KUKA KRL program: f1_Kuka_APT214T02S14.SRC

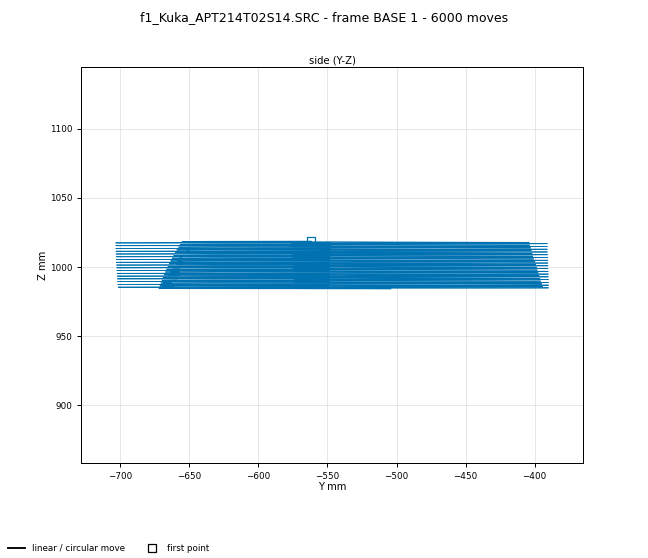
[picture p0: tool path of f1_Kuka_APT214T02S14.SRC in frame BASE 1, 6000 of 6001 moves have a stored position in this frame; points joined in program order, loops and branches not executed]
&ACCESS RVP
&REL 2
&PARAM TEMPLATE = C:\KRC\Roboter\Template\vorgabe
&PARAM EDITMASK = *
DEF f1_Kuka_APT214T02S14()


;FOLD INI;%{PE}%V3.2.0,%MKUKATPBASIS,%CINIT,%VCOMMON,%P
  ;FOLD BAS INI;%{E}%V3.2.0,%MKUKATPBASIS,%CINIT,%VINIT,%P
    GLOBAL INTERRUPT DECL 3 WHEN $STOPMESS==TRUE DO IR_STOPM ( )
    INTERRUPT ON 3
    BAS (#INITMOV,0 )
  ;ENDFOLD (BAS INI)
  ;FOLD USER INI;%{E}%V3.2.0,%MKUKATPUSER,%CINIT,%VINIT,%P
    ;Make your modifications here
  ;ENDFOLD (USER INI)
;ENDFOLD (INI)


;*** Make Null PTP Move
  PTP $pos_act

;*** Auto Load The Correct TOOL Data
  $tool=tool_data[2]

;*** Auto Load The Correct BASE Data
  $base=base_data[1]

  $ADVANCE = 5

;*** Restate Last Velocity
MMPM(30000.0)
SetRPM(8000)
LIN {X -0.057,Y -561.643,Z 1018.748,A 0.000,B 0.000,C 90.000,E1 350.679} C_DIS
LIN {X 0.006,Y -566.271,Z 1018.744,A 0.000,B 0.000,C 90.000,E1 349.982} C_DIS
LIN {X -0.209,Y -569.658,Z 1018.741,A 0.000,B 0.000,C 90.000,E1 349.454} C_DIS
LIN {X 0.145,Y -575.133,Z 1018.736,A 0.000,B 0.000,C 90.000,E1 348.465} C_DIS
LIN {X 0.098,Y -580.048,Z 1018.731,A 0.000,B 0.000,C 90.000,E1 347.521} C_DIS
LIN {X -0.016,Y -582.690,Z 1018.728,A 0.000,B 0.000,C 90.000,E1 346.992} C_DIS
LIN {X -0.106,Y -587.042,Z 1018.723,A 0.000,B 0.000,C 90.000,E1 346.061} C_DIS
LIN {X 0.162,Y -592.851,Z 1018.715,A 0.000,B 0.000,C 90.000,E1 344.700} C_DIS
LIN {X -0.022,Y -596.197,Z 1018.711,A 0.000,B 0.000,C 90.000,E1 343.921} C_DIS
LIN {X 0.114,Y -600.480,Z 1018.705,A 0.000,B 0.000,C 90.000,E1 342.851} C_DIS
LIN {X 0.194,Y -603.554,Z 1018.700,A 0.000,B 0.000,C 90.000,E1 342.054} C_DIS
LIN {X -0.152,Y -607.453,Z 1018.695,A 0.000,B 0.000,C 90.000,E1 341.040} C_DIS
LIN {X 0.011,Y -610.104,Z 1018.690,A 0.000,B 0.000,C 90.000,E1 340.242} C_DIS
LIN {X -0.056,Y -613.405,Z 1018.685,A 0.000,B 0.000,C 90.000,E1 339.209} C_DIS
LIN {X 0.142,Y -616.518,Z 1018.679,A 0.000,B 0.000,C 90.000,E1 338.156} C_DIS
LIN {X 0.387,Y -619.399,Z 1018.673,A 0.000,B 0.000,C 90.000,E1 337.102} C_DIS
LIN {X 0.107,Y -621.483,Z 1018.669,A 0.000,B 0.000,C 90.000,E1 336.357} C_DIS
LIN {X -0.153,Y -624.569,Z 1018.662,A 0.000,B 0.000,C 90.000,E1 335.101} C_DIS
LIN {X -0.110,Y -626.888,Z 1018.656,A 0.000,B 0.000,C 90.000,E1 334.076} C_DIS
LIN {X -0.009,Y -629.345,Z 1018.649,A 0.000,B 0.000,C 90.000,E1 332.794} C_DIS
LIN {X 0.070,Y -630.776,Z 1018.645,A 0.000,B 0.000,C 90.000,E1 332.025} C_DIS
LIN {X 0.010,Y -633.221,Z 1018.636,A 0.000,B 0.000,C 90.000,E1 330.511} C_DIS
LIN {X 0.149,Y -634.686,Z 1018.631,A 0.000,B 0.000,C 90.000,E1 329.488} C_DIS
LIN {X -0.103,Y -636.263,Z 1018.624,A 0.000,B 0.000,C 90.000,E1 328.250} C_DIS
LIN {X 0.259,Y -637.804,Z 1018.615,A 0.000,B 0.000,C 90.000,E1 326.707} C_DIS
LIN {X 0.039,Y -638.702,Z 1018.610,A 0.000,B 0.000,C 90.000,E1 325.722} C_DIS
LIN {X -0.035,Y -639.237,Z 1018.605,A 0.000,B 0.000,C 90.000,E1 324.975} C_DIS
LIN {X 0.163,Y -639.802,Z 1018.599,A 0.000,B 0.000,C 90.000,E1 323.703} C_DIS
LIN {X 0.259,Y -640.219,Z 1018.590,A 0.000,B 0.000,C 90.000,E1 322.190} C_DIS
LIN {X 0.161,Y -640.668,Z 1018.579,A 0.000,B 0.000,C 90.000,E1 320.194} C_DIS
LIN {X -0.417,Y -641.541,Z 1018.568,A 0.000,B 0.000,C 90.000,E1 318.243} C_DIS
LIN {X 0.035,Y -642.135,Z 1018.560,A 0.000,B 0.000,C 90.000,E1 316.701} C_DIS
LIN {X 0.325,Y -643.049,Z 1018.548,A 0.000,B 0.000,C 90.000,E1 314.676} C_DIS
LIN {X -0.126,Y -643.821,Z 1018.540,A 0.000,B 0.000,C 90.000,E1 313.218} C_DIS
LIN {X -0.031,Y -644.445,Z 1018.533,A 0.000,B 0.000,C 90.000,E1 311.962} C_DIS
LIN {X 0.052,Y -645.030,Z 1018.525,A 0.000,B 0.000,C 90.000,E1 310.458} C_DIS
LIN {X -0.187,Y -645.402,Z 1018.519,A 0.000,B 0.000,C 90.000,E1 309.483} C_DIS
LIN {X -0.007,Y -645.815,Z 1018.512,A 0.000,B 0.000,C 90.000,E1 308.222} C_DIS
LIN {X -0.130,Y -645.997,Z 1018.507,A 0.000,B 0.000,C 90.000,E1 307.237} C_DIS
LIN {X 0.087,Y -646.328,Z 1018.499,A 0.000,B 0.000,C 90.000,E1 305.724} C_DIS
LIN {X 0.403,Y -646.825,Z 1018.487,A 0.000,B 0.000,C 90.000,E1 303.706} C_DIS
LIN {X -0.135,Y -649.932,Z 1018.463,A 0.000,B 0.000,C 90.000,E1 299.283} C_DIS
LIN {X -0.198,Y -652.108,Z 1018.452,A 0.000,B 0.000,C 90.000,E1 297.308} C_DIS
LIN {X 0.032,Y -653.582,Z 1018.445,A 0.000,B 0.000,C 90.000,E1 296.052} C_DIS
LIN {X -0.122,Y -654.484,Z 1018.439,A 0.000,B 0.000,C 90.000,E1 295.079} C_DIS
LIN {X 0.046,Y -655.090,Z 1018.434,A 0.000,B 0.000,C 90.000,E1 294.079} C_DIS
LIN {X 0.223,Y -655.267,Z 1018.428,A 0.000,B 0.000,C 90.000,E1 293.078} C_DIS
LIN {X 0.259,Y -655.153,Z 1018.422,A 0.000,B 0.000,C 90.000,E1 291.844} C_DIS
LIN {X 0.363,Y -654.956,Z 1018.420,A 0.000,B 0.000,C 90.000,E1 291.589} C_DIS
LIN {X 0.327,Y -654.216,Z 1018.417,A 0.000,B 0.000,C 90.000,E1 291.099} C_DIS
LIN {X 0.287,Y -652.605,Z 1018.415,A 0.000,B 0.000,C 90.000,E1 290.610} C_DIS
LIN {X 0.150,Y -651.584,Z 1018.413,A 0.000,B 0.000,C 90.000,E1 290.375} C_DIS
LIN {X 0.238,Y -649.491,Z 1018.412,A 0.000,B 0.000,C 90.000,E1 290.120} C_DIS
LIN {X 0.095,Y -647.416,Z 1018.411,A 0.000,B 0.000,C 90.000,E1 289.885} C_DIS
LIN {X -0.373,Y -645.811,Z 1018.410,A 0.000,B 0.000,C 90.000,E1 289.758} C_DIS
LIN {X 0.299,Y -641.940,Z 1018.408,A 0.000,B 0.000,C 90.000,E1 289.450} C_DIS
LIN {X 0.228,Y -639.375,Z 1018.407,A 0.000,B 0.000,C 90.000,E1 289.268} C_DIS
LIN {X -0.172,Y -637.836,Z 1018.407,A 0.000,B 0.000,C 90.000,E1 289.214} C_DIS
LIN {X 0.150,Y -629.654,Z 1018.404,A 0.000,B 0.000,C 90.000,E1 288.779} C_DIS
LIN {X 0.077,Y -622.622,Z 1018.403,A 0.000,B 0.000,C 90.000,E1 288.489} C_DIS
LIN {X 0.244,Y -618.964,Z 1018.402,A 0.000,B 0.000,C 90.000,E1 288.308} C_DIS
LIN {X 0.190,Y -618.908,Z 1018.402,A 0.000,B 0.000,C 90.000,E1 288.308} C_DIS
LIN {X -0.227,Y -624.386,Z 1018.398,A 0.000,B 0.000,C 90.000,E1 287.583} C_DIS
LIN {X 0.131,Y -628.209,Z 1018.395,A 0.000,B 0.000,C 90.000,E1 287.040} C_DIS
LIN {X -0.090,Y -631.728,Z 1018.392,A 0.000,B 0.000,C 90.000,E1 286.551} C_DIS
LIN {X 0.134,Y -635.498,Z 1018.388,A 0.000,B 0.000,C 90.000,E1 285.898} C_DIS
LIN {X -0.045,Y -636.836,Z 1018.387,A 0.000,B 0.000,C 90.000,E1 285.662} C_DIS
LIN {X 0.224,Y -639.214,Z 1018.384,A 0.000,B 0.000,C 90.000,E1 285.134} C_DIS
LIN {X 0.059,Y -640.247,Z 1018.383,A 0.000,B 0.000,C 90.000,E1 284.898} C_DIS
LIN {X 0.359,Y -642.827,Z 1018.379,A 0.000,B 0.000,C 90.000,E1 284.120} C_DIS
LIN {X 0.204,Y -643.554,Z 1018.377,A 0.000,B 0.000,C 90.000,E1 283.883} C_DIS
LIN {X 0.050,Y -644.125,Z 1018.376,A 0.000,B 0.000,C 90.000,E1 283.647} C_DIS
LIN {X -0.251,Y -644.976,Z 1018.373,A 0.000,B 0.000,C 90.000,E1 283.175} C_DIS
LIN {X -0.065,Y -645.862,Z 1018.369,A 0.000,B 0.000,C 90.000,E1 282.411} C_DIS
LIN {X 0.140,Y -646.048,Z 1018.366,A 0.000,B 0.000,C 90.000,E1 281.895} C_DIS
LIN {X -0.148,Y -645.864,Z 1018.363,A 0.000,B 0.000,C 90.000,E1 281.422} C_DIS
LIN {X 0.044,Y -645.078,Z 1018.359,A 0.000,B 0.000,C 90.000,E1 280.658} C_DIS
LIN {X 0.261,Y -644.156,Z 1018.357,A 0.000,B 0.000,C 90.000,E1 280.141} C_DIS
LIN {X -0.048,Y -642.825,Z 1018.354,A 0.000,B 0.000,C 90.000,E1 279.670} C_DIS
LIN {X 0.161,Y -641.128,Z 1018.351,A 0.000,B 0.000,C 90.000,E1 279.151} C_DIS
LIN {X -0.004,Y -640.167,Z 1018.350,A 0.000,B 0.000,C 90.000,E1 278.916} C_DIS
LIN {X 0.191,Y -637.899,Z 1018.347,A 0.000,B 0.000,C 90.000,E1 278.398} C_DIS
LIN {X -0.258,Y -634.856,Z 1018.344,A 0.000,B 0.000,C 90.000,E1 277.936} C_DIS
LIN {X -0.158,Y -630.199,Z 1018.341,A 0.000,B 0.000,C 90.000,E1 277.296} C_DIS
LIN {X 0.115,Y -626.854,Z 1018.338,A 0.000,B 0.000,C 90.000,E1 276.891} C_DIS
LIN {X 0.180,Y -620.711,Z 1018.335,A 0.000,B 0.000,C 90.000,E1 276.258} C_DIS
LIN {X 0.086,Y -613.759,Z 1018.332,A 0.000,B 0.000,C 90.000,E1 275.682} C_DIS
LIN {X -0.147,Y -606.089,Z 1018.329,A 0.000,B 0.000,C 90.000,E1 275.163} C_DIS
LIN {X 0.078,Y -599.683,Z 1018.327,A 0.000,B 0.000,C 90.000,E1 274.759} C_DIS
LIN {X -0.286,Y -594.298,Z 1018.325,A 0.000,B 0.000,C 90.000,E1 274.531} C_DIS
LIN {X -0.227,Y -589.075,Z 1018.324,A 0.000,B 0.000,C 90.000,E1 274.302} C_DIS
LIN {X 0.101,Y -585.655,Z 1018.323,A 0.000,B 0.000,C 90.000,E1 274.131} C_DIS
LIN {X 0.250,Y -577.484,Z 1018.322,A 0.000,B 0.000,C 90.000,E1 273.898} C_DIS
LIN {X 0.081,Y -571.402,Z 1018.321,A 0.000,B 0.000,C 90.000,E1 273.784} C_DIS
LIN {X 0.255,Y -565.128,Z 1018.321,A 0.000,B 0.000,C 90.000,E1 273.669} C_DIS
LIN {X -0.046,Y -559.419,Z 1018.320,A 0.000,B 0.000,C 90.000,E1 273.669} C_DIS
LIN {X -0.087,Y -543.707,Z 1018.320,A 0.000,B 0.000,C 90.000,E1 273.669} C_DIS
LIN {X 0.158,Y -543.322,Z 1018.320,A 0.000,B 0.000,C 90.000,E1 273.555} C_DIS
LIN {X 0.168,Y -542.409,Z 1018.317,A 0.000,B 0.000,C 90.000,E1 273.037} C_DIS
LIN {X 0.219,Y -541.838,Z 1018.314,A 0.000,B 0.000,C 90.000,E1 272.465} C_DIS
LIN {X -0.138,Y -540.755,Z 1018.303,A 0.000,B 0.000,C 90.000,E1 270.516} C_DIS
LIN {X -0.051,Y -540.067,Z 1018.297,A 0.000,B 0.000,C 90.000,E1 269.370} C_DIS
LIN {X 0.022,Y -539.238,Z 1018.290,A 0.000,B 0.000,C 90.000,E1 268.224} C_DIS
LIN {X 0.136,Y -538.155,Z 1018.282,A 0.000,B 0.000,C 90.000,E1 266.788} C_DIS
LIN {X 0.202,Y -537.060,Z 1018.274,A 0.000,B 0.000,C 90.000,E1 265.355} C_DIS
LIN {X -0.198,Y -536.008,Z 1018.266,A 0.000,B 0.000,C 90.000,E1 263.970} C_DIS
LIN {X -0.075,Y -534.864,Z 1018.258,A 0.000,B 0.000,C 90.000,E1 262.527} C_DIS
LIN {X -0.027,Y -533.729,Z 1018.252,A 0.000,B 0.000,C 90.000,E1 261.376} C_DIS
LIN {X 0.162,Y -532.442,Z 1018.246,A 0.000,B 0.000,C 90.000,E1 260.208} C_DIS
LIN {X -0.122,Y -529.887,Z 1018.233,A 0.000,B 0.000,C 90.000,E1 257.937} C_DIS
LIN {X 0.163,Y -528.380,Z 1018.225,A 0.000,B 0.000,C 90.000,E1 256.464} C_DIS
LIN {X -0.113,Y -527.071,Z 1018.219,A 0.000,B 0.000,C 90.000,E1 255.338} C_DIS
LIN {X 0.112,Y -525.448,Z 1018.211,A 0.000,B 0.000,C 90.000,E1 253.866} C_DIS
LIN {X 0.089,Y -523.580,Z 1018.201,A 0.000,B 0.000,C 90.000,E1 252.127} C_DIS
LIN {X -0.103,Y -522.648,Z 1018.196,A 0.000,B 0.000,C 90.000,E1 251.275} C_DIS
LIN {X -0.173,Y -520.803,Z 1018.188,A 0.000,B 0.000,C 90.000,E1 249.826} C_DIS
LIN {X 0.037,Y -518.472,Z 1018.178,A 0.000,B 0.000,C 90.000,E1 248.050} C_DIS
LIN {X -0.090,Y -516.086,Z 1018.168,A 0.000,B 0.000,C 90.000,E1 246.305} C_DIS
LIN {X 0.166,Y -514.407,Z 1018.162,A 0.000,B 0.000,C 90.000,E1 245.101} C_DIS
LIN {X -0.062,Y -512.631,Z 1018.155,A 0.000,B 0.000,C 90.000,E1 243.948} C_DIS
LIN {X 0.143,Y -510.808,Z 1018.149,A 0.000,B 0.000,C 90.000,E1 242.743} C_DIS
LIN {X 0.149,Y -507.336,Z 1018.137,A 0.000,B 0.000,C 90.000,E1 240.667} C_DIS
LIN {X 0.050,Y -505.272,Z 1018.131,A 0.000,B 0.000,C 90.000,E1 239.488} C_DIS
LIN {X -0.134,Y -503.619,Z 1018.126,A 0.000,B 0.000,C 90.000,E1 238.614} C_DIS
LIN {X 0.136,Y -500.140,Z 1018.116,A 0.000,B 0.000,C 90.000,E1 236.786} C_DIS
LIN {X -0.092,Y -496.781,Z 1018.107,A 0.000,B 0.000,C 90.000,E1 235.308} C_DIS
LIN {X 0.047,Y -495.422,Z 1018.104,A 0.000,B 0.000,C 90.000,E1 234.689} C_DIS
LIN {X -0.260,Y -491.789,Z 1018.096,A 0.000,B 0.000,C 90.000,E1 233.210} C_DIS
LIN {X -0.041,Y -488.114,Z 1018.087,A 0.000,B 0.000,C 90.000,E1 231.662} C_DIS
LIN {X -0.062,Y -483.890,Z 1018.077,A 0.000,B 0.000,C 90.000,E1 229.828} C_DIS
LIN {X -0.319,Y -478.333,Z 1018.063,A 0.000,B 0.000,C 90.000,E1 227.391} C_DIS
LIN {X -0.011,Y -472.530,Z 1018.048,A 0.000,B 0.000,C 90.000,E1 224.555} C_DIS
LIN {X -0.056,Y -467.938,Z 1018.035,A 0.000,B 0.000,C 90.000,E1 222.366} C_DIS
LIN {X 0.069,Y -464.045,Z 1018.025,A 0.000,B 0.000,C 90.000,E1 220.458} C_DIS
LIN {X 0.019,Y -461.289,Z 1018.018,A 0.000,B 0.000,C 90.000,E1 219.197} C_DIS
LIN {X -0.075,Y -458.413,Z 1018.011,A 0.000,B 0.000,C 90.000,E1 217.935} C_DIS
LIN {X 0.041,Y -452.716,Z 1017.997,A 0.000,B 0.000,C 90.000,E1 215.358} C_DIS
LIN {X -0.070,Y -450.612,Z 1017.991,A 0.000,B 0.000,C 90.000,E1 214.405} C_DIS
LIN {X 0.126,Y -447.787,Z 1017.984,A 0.000,B 0.000,C 90.000,E1 213.086} C_DIS
LIN {X 0.095,Y -444.243,Z 1017.975,A 0.000,B 0.000,C 90.000,E1 211.465} C_DIS
LIN {X -0.058,Y -441.474,Z 1017.968,A 0.000,B 0.000,C 90.000,E1 210.178} C_DIS
LIN {X -0.062,Y -437.774,Z 1017.959,A 0.000,B 0.000,C 90.000,E1 208.537} C_DIS
LIN {X -0.126,Y -432.502,Z 1017.946,A 0.000,B 0.000,C 90.000,E1 206.232} C_DIS
LIN {X 0.073,Y -427.990,Z 1017.935,A 0.000,B 0.000,C 90.000,E1 204.207} C_DIS
LIN {X 0.168,Y -422.799,Z 1017.922,A 0.000,B 0.000,C 90.000,E1 201.844} C_DIS
LIN {X 0.122,Y -417.466,Z 1017.906,A 0.000,B 0.000,C 90.000,E1 199.141} C_DIS
LIN {X -0.105,Y -412.615,Z 1017.891,A 0.000,B 0.000,C 90.000,E1 196.441} C_DIS
LIN {X 0.195,Y -408.358,Z 1017.876,A 0.000,B 0.000,C 90.000,E1 193.647} C_DIS
LIN {X 0.070,Y -404.749,Z 1017.861,A 0.000,B 0.000,C 90.000,E1 190.894} C_DIS
LIN {X 0.084,Y -404.194,Z 1017.857,A 0.000,B 0.000,C 90.000,E1 190.197} C_DIS
LIN {X 0.093,Y -404.018,Z 1017.853,A 0.000,B 0.000,C 90.000,E1 189.500} C_DIS
LIN {X 0.097,Y -404.430,Z 1017.851,A 0.000,B 0.000,C 90.000,E1 189.151} C_DIS
LIN {X 0.192,Y -404.984,Z 1017.847,A 0.000,B 0.000,C 90.000,E1 188.454} C_DIS
LIN {X 0.198,Y -405.583,Z 1017.845,A 0.000,B 0.000,C 90.000,E1 188.106} C_DIS
LIN {X 0.121,Y -407.332,Z 1017.842,A 0.000,B 0.000,C 90.000,E1 187.530} C_DIS
LIN {X 0.118,Y -409.450,Z 1017.839,A 0.000,B 0.000,C 90.000,E1 187.011} C_DIS
LIN {X -0.044,Y -413.526,Z 1017.835,A 0.000,B 0.000,C 90.000,E1 186.258} C_DIS
LIN {X -0.010,Y -416.959,Z 1017.832,A 0.000,B 0.000,C 90.000,E1 185.739} C_DIS
LIN {X 0.062,Y -423.247,Z 1017.827,A 0.000,B 0.000,C 90.000,E1 184.878} C_DIS
LIN {X 0.138,Y -436.886,Z 1017.818,A 0.000,B 0.000,C 90.000,E1 183.212} C_DIS
LIN {X 0.195,Y -443.636,Z 1017.814,A 0.000,B 0.000,C 90.000,E1 182.407} C_DIS
LIN {X 0.161,Y -455.608,Z 1017.806,A 0.000,B 0.000,C 90.000,E1 180.974} C_DIS
LIN {X -0.192,Y -463.235,Z 1017.800,A 0.000,B 0.000,C 90.000,E1 180.057} C_DIS
LIN {X -0.229,Y -471.737,Z 1017.794,A 0.000,B 0.000,C 90.000,E1 178.969} C_DIS
LIN {X 0.081,Y -478.889,Z 1017.789,A 0.000,B 0.000,C 90.000,E1 177.993} C_DIS
LIN {X 0.129,Y -486.902,Z 1017.783,A 0.000,B 0.000,C 90.000,E1 176.906} C_DIS
LIN {X -0.153,Y -494.425,Z 1017.777,A 0.000,B 0.000,C 90.000,E1 175.869} C_DIS
LIN {X 0.120,Y -501.615,Z 1017.771,A 0.000,B 0.000,C 90.000,E1 174.780} C_DIS
LIN {X -0.177,Y -509.345,Z 1017.765,A 0.000,B 0.000,C 90.000,E1 173.628} C_DIS
LIN {X 0.106,Y -516.789,Z 1017.758,A 0.000,B 0.000,C 90.000,E1 172.413} C_DIS
LIN {X -0.007,Y -523.522,Z 1017.751,A 0.000,B 0.000,C 90.000,E1 171.254} C_DIS
LIN {X -0.241,Y -525.133,Z 1017.750,A 0.000,B 0.000,C 90.000,E1 171.027} C_DIS
LIN {X 0.004,Y -538.475,Z 1017.737,A 0.000,B 0.000,C 90.000,E1 168.701} C_DIS
LIN {X 0.212,Y -543.433,Z 1017.733,A 0.000,B 0.000,C 90.000,E1 167.825} C_DIS
LIN {X 0.271,Y -551.310,Z 1017.725,A 0.000,B 0.000,C 90.000,E1 166.408} C_DIS
LIN {X 0.072,Y -558.306,Z 1017.718,A 0.000,B 0.000,C 90.000,E1 165.172} C_DIS
LIN {X 0.123,Y -565.030,Z 1017.711,A 0.000,B 0.000,C 90.000,E1 163.921} C_DIS
LIN {X -0.219,Y -568.632,Z 1017.707,A 0.000,B 0.000,C 90.000,E1 163.268} C_DIS
LIN {X -0.290,Y -574.124,Z 1017.701,A 0.000,B 0.000,C 90.000,E1 162.181} C_DIS
LIN {X 0.079,Y -578.114,Z 1017.696,A 0.000,B 0.000,C 90.000,E1 161.329} C_DIS
LIN {X 0.075,Y -583.755,Z 1017.690,A 0.000,B 0.000,C 90.000,E1 160.115} C_DIS
LIN {X 0.212,Y -588.411,Z 1017.684,A 0.000,B 0.000,C 90.000,E1 159.028} C_DIS
LIN {X -0.040,Y -593.946,Z 1017.676,A 0.000,B 0.000,C 90.000,E1 157.720} C_DIS
LIN {X 0.080,Y -596.018,Z 1017.673,A 0.000,B 0.000,C 90.000,E1 157.177} C_DIS
LIN {X 0.276,Y -599.849,Z 1017.667,A 0.000,B 0.000,C 90.000,E1 156.102} C_DIS
LIN {X -0.198,Y -602.527,Z 1017.663,A 0.000,B 0.000,C 90.000,E1 155.357} C_DIS
LIN {X 0.037,Y -606.641,Z 1017.656,A 0.000,B 0.000,C 90.000,E1 154.024} C_DIS
LIN {X -0.204,Y -610.468,Z 1017.648,A 0.000,B 0.000,C 90.000,E1 152.743} C_DIS
LIN {X -0.066,Y -613.353,Z 1017.643,A 0.000,B 0.000,C 90.000,E1 151.691} C_DIS
LIN {X 0.097,Y -616.826,Z 1017.636,A 0.000,B 0.000,C 90.000,E1 150.383} C_DIS
LIN {X 0.072,Y -621.488,Z 1017.626,A 0.000,B 0.000,C 90.000,E1 148.584} C_DIS
LIN {X 0.150,Y -625.467,Z 1017.617,A 0.000,B 0.000,C 90.000,E1 147.041} C_DIS
LIN {X -0.231,Y -628.672,Z 1017.610,A 0.000,B 0.000,C 90.000,E1 145.801} C_DIS
LIN {X 0.165,Y -633.185,Z 1017.600,A 0.000,B 0.000,C 90.000,E1 143.989} C_DIS
LIN {X -0.240,Y -636.337,Z 1017.593,A 0.000,B 0.000,C 90.000,E1 142.763} C_DIS
LIN {X -0.088,Y -638.835,Z 1017.587,A 0.000,B 0.000,C 90.000,E1 141.743} C_DIS
LIN {X -0.007,Y -642.582,Z 1017.579,A 0.000,B 0.000,C 90.000,E1 140.231} C_DIS
LIN {X 0.054,Y -646.249,Z 1017.571,A 0.000,B 0.000,C 90.000,E1 138.728} C_DIS
LIN {X -0.024,Y -651.841,Z 1017.558,A 0.000,B 0.000,C 90.000,E1 136.500} C_DIS
LIN {X 0.151,Y -656.550,Z 1017.549,A 0.000,B 0.000,C 90.000,E1 134.757} C_DIS
LIN {X -0.043,Y -661.721,Z 1017.539,A 0.000,B 0.000,C 90.000,E1 133.056} C_DIS
LIN {X -0.081,Y -665.591,Z 1017.532,A 0.000,B 0.000,C 90.000,E1 131.838} C_DIS
LIN {X -0.047,Y -668.544,Z 1017.527,A 0.000,B 0.000,C 90.000,E1 130.862} C_DIS
LIN {X 0.030,Y -671.481,Z 1017.522,A 0.000,B 0.000,C 90.000,E1 129.886} C_DIS
LIN {X -0.262,Y -675.615,Z 1017.514,A 0.000,B 0.000,C 90.000,E1 128.463} C_DIS
LIN {X 0.028,Y -678.946,Z 1017.507,A 0.000,B 0.000,C 90.000,E1 127.237} C_DIS
LIN {X -0.014,Y -682.823,Z 1017.499,A 0.000,B 0.000,C 90.000,E1 125.804} C_DIS
LIN {X -0.010,Y -686.062,Z 1017.492,A 0.000,B 0.000,C 90.000,E1 124.612} C_DIS
LIN {X -0.176,Y -687.897,Z 1017.488,A 0.000,B 0.000,C 90.000,E1 123.913} C_DIS
LIN {X 0.113,Y -691.502,Z 1017.480,A 0.000,B 0.000,C 90.000,E1 122.467} C_DIS
LIN {X 0.090,Y -694.461,Z 1017.474,A 0.000,B 0.000,C 90.000,E1 121.288} C_DIS
LIN {X -0.117,Y -697.082,Z 1017.467,A 0.000,B 0.000,C 90.000,E1 120.129} C_DIS
LIN {X 0.046,Y -698.438,Z 1017.463,A 0.000,B 0.000,C 90.000,E1 119.411} C_DIS
LIN {X 0.147,Y -700.214,Z 1017.457,A 0.000,B 0.000,C 90.000,E1 118.231} C_DIS
LIN {X 0.342,Y -701.001,Z 1017.453,A 0.000,B 0.000,C 90.000,E1 117.513} C_DIS
LIN {X -0.307,Y -702.750,Z 1017.441,A 0.000,B 0.000,C 90.000,E1 115.463} C_DIS
LIN {X 0.237,Y -703.225,Z 1017.438,A 0.000,B 0.000,C 90.000,E1 114.719} C_DIS
LIN {X 0.158,Y -703.239,Z 1017.435,A 0.000,B 0.000,C 90.000,E1 114.259} C_DIS
LIN {X 0.150,Y -703.096,Z 1017.434,A 0.000,B 0.000,C 90.000,E1 114.027} C_DIS
LIN {X 0.065,Y -702.357,Z 1017.431,A 0.000,B 0.000,C 90.000,E1 113.567} C_DIS
LIN {X 0.061,Y -701.548,Z 1017.430,A 0.000,B 0.000,C 90.000,E1 113.334} C_DIS
LIN {X -0.315,Y -699.027,Z 1017.427,A 0.000,B 0.000,C 90.000,E1 112.898} C_DIS
LIN {X -0.183,Y -698.177,Z 1017.426,A 0.000,B 0.000,C 90.000,E1 112.770} C_DIS
LIN {X -0.051,Y -696.915,Z 1017.426,A 0.000,B 0.000,C 90.000,E1 112.642} C_DIS
LIN {X 0.256,Y -690.392,Z 1017.424,A 0.000,B 0.000,C 90.000,E1 112.206} C_DIS
LIN {X -0.206,Y -688.443,Z 1017.423,A 0.000,B 0.000,C 90.000,E1 112.153} C_DIS
LIN {X 0.230,Y -685.655,Z 1017.423,A 0.000,B 0.000,C 90.000,E1 112.025} C_DIS
LIN {X 0.192,Y -683.468,Z 1017.422,A 0.000,B 0.000,C 90.000,E1 111.972} C_DIS
LIN {X -0.229,Y -675.140,Z 1017.422,A 0.000,B 0.000,C 90.000,E1 111.897} C_DIS
LIN {X -0.243,Y -615.838,Z 1017.422,A 0.000,B 0.000,C 90.000,E1 111.897} C_DIS
LIN {X 0.286,Y -610.721,Z 1017.421,A 0.000,B 0.000,C 90.000,E1 111.716} C_DIS
LIN {X 0.239,Y -605.536,Z 1017.420,A 0.000,B 0.000,C 90.000,E1 111.535} C_DIS
LIN {X -0.193,Y -599.101,Z 1017.418,A 0.000,B 0.000,C 90.000,E1 111.280} C_DIS
LIN {X -0.045,Y -593.333,Z 1017.416,A 0.000,B 0.000,C 90.000,E1 110.918} C_DIS
LIN {X 0.263,Y -587.741,Z 1017.414,A 0.000,B 0.000,C 90.000,E1 110.482} C_DIS
LIN {X 0.180,Y -576.703,Z 1017.409,A 0.000,B 0.000,C 90.000,E1 109.577} C_DIS
LIN {X 0.101,Y -570.755,Z 1017.406,A 0.000,B 0.000,C 90.000,E1 109.141} C_DIS
LIN {X 0.059,Y -562.295,Z 1017.404,A 0.000,B 0.000,C 90.000,E1 108.671} C_DIS
LIN {X -0.267,Y -555.586,Z 1017.402,A 0.000,B 0.000,C 90.000,E1 108.362} C_DIS
LIN {X -0.040,Y -549.719,Z 1017.400,A 0.000,B 0.000,C 90.000,E1 108.000} C_DIS
LIN {X 0.141,Y -548.390,Z 1017.399,A 0.000,B 0.000,C 90.000,E1 107.819} C_DIS
LIN {X 0.099,Y -548.381,Z 1017.399,A 0.000,B 0.000,C 90.000,E1 107.819} C_DIS
LIN {X 0.096,Y -548.038,Z 1017.397,A 0.000,B 0.000,C 90.000,E1 107.402} C_DIS
LIN {X 0.126,Y -548.283,Z 1017.392,A 0.000,B 0.000,C 90.000,E1 106.567} C_DIS
LIN {X -0.047,Y -549.100,Z 1017.383,A 0.000,B 0.000,C 90.000,E1 104.898} C_DIS
LIN {X 0.021,Y -551.619,Z 1017.363,A 0.000,B 0.000,C 90.000,E1 101.243} C_DIS
LIN {X -0.218,Y -553.984,Z 1017.350,A 0.000,B 0.000,C 90.000,E1 99.029} C_DIS
LIN {X 0.065,Y -554.939,Z 1017.345,A 0.000,B 0.000,C 90.000,E1 98.163} C_DIS
LIN {X 0.113,Y -556.784,Z 1017.336,A 0.000,B 0.000,C 90.000,E1 96.486} C_DIS
LIN {X -0.063,Y -557.848,Z 1017.330,A 0.000,B 0.000,C 90.000,E1 95.391} C_DIS
LIN {X -0.271,Y -558.743,Z 1017.324,A 0.000,B 0.000,C 90.000,E1 94.302} C_DIS
LIN {X 0.217,Y -559.593,Z 1017.316,A 0.000,B 0.000,C 90.000,E1 92.865} C_DIS
LIN {X 0.217,Y -560.345,Z 1017.307,A 0.000,B 0.000,C 90.000,E1 91.203} C_DIS
LIN {X 0.225,Y -561.031,Z 1017.298,A 0.000,B 0.000,C 90.000,E1 89.542} C_DIS
LIN {X 0.163,Y -561.609,Z 1017.290,A 0.000,B 0.000,C 90.000,E1 88.165} C_DIS
LIN {X -0.009,Y -561.906,Z 1017.284,A 0.000,B 0.000,C 90.000,E1 87.078} C_DIS
LIN {X 0.065,Y -562.206,Z 1017.275,A 0.000,B 0.000,C 90.000,E1 85.412} C_DIS
LIN {X 0.199,Y -562.545,Z 1017.265,A 0.000,B 0.000,C 90.000,E1 83.742} C_DIS
LIN {X 0.104,Y -562.770,Z 1017.259,A 0.000,B 0.000,C 90.000,E1 82.648} C_DIS
LIN {X -0.085,Y -563.293,Z 1017.249,A 0.000,B 0.000,C 90.000,E1 80.735} C_DIS
LIN {X -0.002,Y -564.091,Z 1017.236,A 0.000,B 0.000,C 90.000,E1 78.522} C_DIS
LIN {X -0.118,Y -564.947,Z 1017.227,A 0.000,B 0.000,C 90.000,E1 76.881} C_DIS
LIN {X -0.157,Y -566.331,Z 1017.215,A 0.000,B 0.000,C 90.000,E1 74.685} C_DIS
LIN {X 0.060,Y -567.604,Z 1017.206,A 0.000,B 0.000,C 90.000,E1 73.015} C_DIS
LIN {X 0.129,Y -568.610,Z 1017.198,A 0.000,B 0.000,C 90.000,E1 71.638} C_DIS
LIN {X 0.010,Y -569.824,Z 1017.189,A 0.000,B 0.000,C 90.000,E1 70.007} C_DIS
LIN {X -0.079,Y -571.122,Z 1017.178,A 0.000,B 0.000,C 90.000,E1 68.103} C_DIS
LIN {X 0.076,Y -572.215,Z 1017.168,A 0.000,B 0.000,C 90.000,E1 66.177} C_DIS
LIN {X 0.129,Y -572.934,Z 1017.159,A 0.000,B 0.000,C 90.000,E1 64.537} C_DIS
LIN {X -0.064,Y -573.642,Z 1017.150,A 0.000,B 0.000,C 90.000,E1 62.922} C_DIS
LIN {X -0.237,Y -574.211,Z 1017.141,A 0.000,B 0.000,C 90.000,E1 61.307} C_DIS
LIN {X 0.032,Y -574.642,Z 1017.133,A 0.000,B 0.000,C 90.000,E1 59.921} C_DIS
LIN {X 0.306,Y -575.026,Z 1017.125,A 0.000,B 0.000,C 90.000,E1 58.535} C_DIS
LIN {X 0.369,Y -575.476,Z 1017.115,A 0.000,B 0.000,C 90.000,E1 56.628} C_DIS
LIN {X -0.161,Y -575.630,Z 1017.109,A 0.000,B 0.000,C 90.000,E1 55.595} C_DIS
LIN {X 0.262,Y -575.723,Z 1017.101,A 0.000,B 0.000,C 90.000,E1 54.196} C_DIS
LIN {X 0.215,Y -575.521,Z 1017.094,A 0.000,B 0.000,C 90.000,E1 52.844} C_DIS
LIN {X 0.007,Y -575.182,Z 1017.088,A 0.000,B 0.000,C 90.000,E1 51.778} C_DIS
LIN {X -0.299,Y -574.711,Z 1017.082,A 0.000,B 0.000,C 90.000,E1 50.723} C_DIS
LIN {X -0.026,Y -573.879,Z 1017.074,A 0.000,B 0.000,C 90.000,E1 49.337} C_DIS
LIN {X 0.030,Y -573.027,Z 1017.068,A 0.000,B 0.000,C 90.000,E1 48.243} C_DIS
LIN {X 0.379,Y -572.281,Z 1017.064,A 0.000,B 0.000,C 90.000,E1 47.391} C_DIS
LIN {X -0.092,Y -571.368,Z 1017.059,A 0.000,B 0.000,C 90.000,E1 46.620} C_DIS
LIN {X -0.177,Y -570.266,Z 1017.054,A 0.000,B 0.000,C 90.000,E1 45.810} C_DIS
LIN {X -0.272,Y -568.999,Z 1017.050,A 0.000,B 0.000,C 90.000,E1 45.000} C_DIS
LIN {X 0.017,Y -567.525,Z 1017.045,A 0.000,B 0.000,C 90.000,E1 44.150} C_DIS
LIN {X -0.017,Y -565.356,Z 1017.039,A 0.000,B 0.000,C 90.000,E1 43.056} C_DIS
LIN {X -0.136,Y -563.436,Z 1017.035,A 0.000,B 0.000,C 90.000,E1 42.243} C_DIS
LIN {X 0.108,Y -561.232,Z 1017.030,A 0.000,B 0.000,C 90.000,E1 41.391} C_DIS
LIN {X -0.131,Y -559.651,Z 1017.027,A 0.000,B 0.000,C 90.000,E1 40.862} C_DIS
LIN {X 0.066,Y -556.969,Z 1017.022,A 0.000,B 0.000,C 90.000,E1 40.011} C_DIS
LIN {X -0.054,Y -553.052,Z 1017.016,A 0.000,B 0.000,C 90.000,E1 38.910} C_DIS
LIN {X -0.286,Y -549.604,Z 1017.012,A 0.000,B 0.000,C 90.000,E1 38.096} C_DIS
LIN {X 0.065,Y -545.262,Z 1017.006,A 0.000,B 0.000,C 90.000,E1 37.076} C_DIS
LIN {X 0.170,Y -541.278,Z 1017.001,A 0.000,B 0.000,C 90.000,E1 36.217} C_DIS
LIN {X 0.068,Y -537.713,Z 1016.997,A 0.000,B 0.000,C 90.000,E1 35.518} C_DIS
LIN {X -0.068,Y -532.390,Z 1016.992,A 0.000,B 0.000,C 90.000,E1 34.532} C_DIS
LIN {X 0.166,Y -526.623,Z 1016.986,A 0.000,B 0.000,C 90.000,E1 33.499} C_DIS
LIN {X 0.205,Y -521.290,Z 1016.981,A 0.000,B 0.000,C 90.000,E1 32.625} C_DIS
LIN {X -0.080,Y -516.572,Z 1016.977,A 0.000,B 0.000,C 90.000,E1 31.926} C_DIS
LIN {X 0.029,Y -511.474,Z 1016.973,A 0.000,B 0.000,C 90.000,E1 31.180} C_DIS
LIN {X -0.174,Y -505.839,Z 1016.969,A 0.000,B 0.000,C 90.000,E1 30.463} C_DIS
LIN {X -0.040,Y -502.296,Z 1016.967,A 0.000,B 0.000,C 90.000,E1 30.001} C_DIS
LIN {X -0.243,Y -495.735,Z 1016.963,A 0.000,B 0.000,C 90.000,E1 29.283} C_DIS
LIN {X 0.300,Y -489.057,Z 1016.958,A 0.000,B 0.000,C 90.000,E1 28.487} C_DIS
LIN {X -0.303,Y -481.950,Z 1016.955,A 0.000,B 0.000,C 90.000,E1 27.847} C_DIS
LIN {X -0.114,Y -474.732,Z 1016.951,A 0.000,B 0.000,C 90.000,E1 27.129} C_DIS
LIN {X -0.065,Y -467.441,Z 1016.947,A 0.000,B 0.000,C 90.000,E1 26.437} C_DIS
LIN {X -0.132,Y -459.951,Z 1016.943,A 0.000,B 0.000,C 90.000,E1 25.771} C_DIS
LIN {X -0.031,Y -449.306,Z 1016.938,A 0.000,B 0.000,C 90.000,E1 24.847} C_DIS
LIN {X 0.109,Y -431.519,Z 1016.929,A 0.000,B 0.000,C 90.000,E1 23.281} C_DIS
LIN {X 0.162,Y -418.312,Z 1016.923,A 0.000,B 0.000,C 90.000,E1 22.025} C_DIS
LIN {X -0.032,Y -406.782,Z 1016.916,A 0.000,B 0.000,C 90.000,E1 20.844} C_DIS
LIN {X 0.060,Y -397.678,Z 1016.910,A 0.000,B 0.000,C 90.000,E1 19.758} C_DIS
LIN {X -0.150,Y -394.148,Z 1016.907,A 0.000,B 0.000,C 90.000,E1 19.268} C_DIS
LIN {X 0.112,Y -392.358,Z 1016.905,A 0.000,B 0.000,C 90.000,E1 18.852} C_DIS
LIN {X -0.179,Y -391.201,Z 1016.902,A 0.000,B 0.000,C 90.000,E1 18.362} C_DIS
LIN {X -0.084,Y -390.894,Z 1016.898,A 0.000,B 0.000,C 90.000,E1 17.638} C_DIS
LIN {X 0.064,Y -391.921,Z 1016.890,A 0.000,B 0.000,C 90.000,E1 16.205} C_DIS
LIN {X 0.145,Y -397.228,Z 1016.865,A 0.000,B 0.000,C 90.000,E1 11.591} C_DIS
LIN {X -0.034,Y -404.136,Z 1016.841,A 0.000,B 0.000,C 90.000,E1 7.409} C_DIS
LIN {X -0.135,Y -412.095,Z 1016.820,A 0.000,B 0.000,C 90.000,E1 3.612} C_DIS
LIN {X -0.119,Y -414.440,Z 1016.814,A 0.000,B 0.000,C 90.000,E1 2.579} C_DIS
LIN {X -0.113,Y -415.372,Z 1016.812,A 0.000,B 0.000,C 90.000,E1 2.236} C_DIS
LIN {X -0.083,Y -417.071,Z 1016.810,A 0.000,B 0.000,C 90.000,E1 1.718} C_DIS
LIN {X -0.096,Y -418.967,Z 1016.808,A 0.000,B 0.000,C 90.000,E1 1.375} C_DIS
LIN {X -0.140,Y -420.859,Z 1016.806,A 0.000,B 0.000,C 90.000,E1 1.088} C_DIS
LIN {X 0.203,Y -423.348,Z 1016.804,A 0.000,B 0.000,C 90.000,E1 0.745} C_DIS
LIN {X -0.201,Y -426.872,Z 1016.803,A 0.000,B 0.000,C 90.000,E1 0.516} C_DIS
LIN {X 0.135,Y -428.624,Z 1016.802,A 0.000,B 0.000,C 90.000,E1 0.344} C_DIS
LIN {X 0.166,Y -438.310,Z 1016.799,A 0.000,B 0.000,C 90.000,E1 359.771} C_DIS
LIN {X -0.002,Y -448.310,Z 1016.796,A 0.000,B 0.000,C 90.000,E1 359.198} C_DIS
LIN {X -0.135,Y -463.144,Z 1016.791,A 0.000,B 0.000,C 90.000,E1 358.339} C_DIS
LIN {X -0.158,Y -479.788,Z 1016.785,A 0.000,B 0.000,C 90.000,E1 357.364} C_DIS
LIN {X 0.124,Y -488.025,Z 1016.783,A 0.000,B 0.000,C 90.000,E1 356.849} C_DIS
LIN {X 0.064,Y -497.732,Z 1016.779,A 0.000,B 0.000,C 90.000,E1 356.274} C_DIS
LIN {X -0.069,Y -508.895,Z 1016.775,A 0.000,B 0.000,C 90.000,E1 355.584} C_DIS
LIN {X -0.205,Y -516.587,Z 1016.773,A 0.000,B 0.000,C 90.000,E1 355.065} C_DIS
LIN {X 0.108,Y -525.380,Z 1016.769,A 0.000,B 0.000,C 90.000,E1 354.375} C_DIS
LIN {X -0.073,Y -532.612,Z 1016.766,A 0.000,B 0.000,C 90.000,E1 353.799} C_DIS
LIN {X 0.028,Y -539.584,Z 1016.762,A 0.000,B 0.000,C 90.000,E1 353.166} C_DIS
LIN {X -0.072,Y -546.155,Z 1016.758,A 0.000,B 0.000,C 90.000,E1 352.527} C_DIS
LIN {X -0.030,Y -552.325,Z 1016.755,A 0.000,B 0.000,C 90.000,E1 351.837} C_DIS
LIN {X 0.205,Y -556.967,Z 1016.752,A 0.000,B 0.000,C 90.000,E1 351.254} C_DIS
LIN {X 0.141,Y -562.117,Z 1016.748,A 0.000,B 0.000,C 90.000,E1 350.566} C_DIS
LIN {X -0.104,Y -565.875,Z 1016.745,A 0.000,B 0.000,C 90.000,E1 350.038} C_DIS
LIN {X 0.238,Y -569.316,Z 1016.742,A 0.000,B 0.000,C 90.000,E1 349.454} C_DIS
LIN {X 0.009,Y -574.835,Z 1016.736,A 0.000,B 0.000,C 90.000,E1 348.522} C_DIS
LIN {X 0.186,Y -578.468,Z 1016.733,A 0.000,B 0.000,C 90.000,E1 347.825} C_DIS
LIN {X -0.155,Y -582.494,Z 1016.728,A 0.000,B 0.000,C 90.000,E1 347.048} C_DIS
LIN {X -0.246,Y -586.907,Z 1016.723,A 0.000,B 0.000,C 90.000,E1 346.117} C_DIS
LIN {X 0.022,Y -592.757,Z 1016.715,A 0.000,B 0.000,C 90.000,E1 344.755} C_DIS
LIN {X -0.161,Y -596.162,Z 1016.711,A 0.000,B 0.000,C 90.000,E1 343.976} C_DIS
LIN {X -0.024,Y -600.456,Z 1016.705,A 0.000,B 0.000,C 90.000,E1 342.906} C_DIS
LIN {X -0.223,Y -604.526,Z 1016.699,A 0.000,B 0.000,C 90.000,E1 341.873} C_DIS
LIN {X -0.286,Y -607.497,Z 1016.695,A 0.000,B 0.000,C 90.000,E1 341.094} C_DIS
LIN {X -0.120,Y -610.185,Z 1016.690,A 0.000,B 0.000,C 90.000,E1 340.296} C_DIS
LIN {X -0.183,Y -613.504,Z 1016.685,A 0.000,B 0.000,C 90.000,E1 339.263} C_DIS
LIN {X -0.209,Y -616.663,Z 1016.679,A 0.000,B 0.000,C 90.000,E1 338.230} C_DIS
LIN {X 0.031,Y -619.602,Z 1016.673,A 0.000,B 0.000,C 90.000,E1 337.177} C_DIS
LIN {X -0.261,Y -622.332,Z 1016.668,A 0.000,B 0.000,C 90.000,E1 336.177} C_DIS
LIN {X 0.310,Y -624.805,Z 1016.662,A 0.000,B 0.000,C 90.000,E1 335.101} C_DIS
LIN {X 0.098,Y -627.703,Z 1016.655,A 0.000,B 0.000,C 90.000,E1 333.845} C_DIS
LIN {X 0.179,Y -629.640,Z 1016.649,A 0.000,B 0.000,C 90.000,E1 332.820} C_DIS
LIN {X 0.023,Y -631.531,Z 1016.643,A 0.000,B 0.000,C 90.000,E1 331.820} C_DIS
LIN {X 0.187,Y -633.576,Z 1016.636,A 0.000,B 0.000,C 90.000,E1 330.539} C_DIS
LIN {X 0.095,Y -635.065,Z 1016.631,A 0.000,B 0.000,C 90.000,E1 329.537} C_DIS
LIN {X 0.064,Y -636.699,Z 1016.624,A 0.000,B 0.000,C 90.000,E1 328.280} C_DIS
LIN {X 0.352,Y -637.784,Z 1016.618,A 0.000,B 0.000,C 90.000,E1 327.248} C_DIS
LIN {X -0.224,Y -638.789,Z 1016.613,A 0.000,B 0.000,C 90.000,E1 326.294} C_DIS
LIN {X 0.095,Y -639.641,Z 1016.607,A 0.000,B 0.000,C 90.000,E1 325.261} C_DIS
LIN {X -0.101,Y -640.181,Z 1016.602,A 0.000,B 0.000,C 90.000,E1 324.276} C_DIS
LIN {X 0.110,Y -640.656,Z 1016.595,A 0.000,B 0.000,C 90.000,E1 323.004} C_DIS
LIN {X 0.209,Y -640.948,Z 1016.588,A 0.000,B 0.000,C 90.000,E1 321.743} C_DIS
LIN {X 0.027,Y -641.698,Z 1016.574,A 0.000,B 0.000,C 90.000,E1 319.256} C_DIS
LIN {X 0.004,Y -642.426,Z 1016.565,A 0.000,B 0.000,C 90.000,E1 317.757} C_DIS
LIN {X 0.089,Y -642.986,Z 1016.558,A 0.000,B 0.000,C 90.000,E1 316.500} C_DIS
LIN {X -0.115,Y -644.058,Z 1016.546,A 0.000,B 0.000,C 90.000,E1 314.271} C_DIS
LIN {X 0.065,Y -644.611,Z 1016.540,A 0.000,B 0.000,C 90.000,E1 313.257} C_DIS
LIN {X 0.111,Y -645.348,Z 1016.532,A 0.000,B 0.000,C 90.000,E1 311.757} C_DIS
LIN {X 0.221,Y -646.005,Z 1016.524,A 0.000,B 0.000,C 90.000,E1 310.253} C_DIS
LIN {X -0.143,Y -646.629,Z 1016.514,A 0.000,B 0.000,C 90.000,E1 308.543} C_DIS
LIN {X 0.144,Y -646.864,Z 1016.509,A 0.000,B 0.000,C 90.000,E1 307.523} C_DIS
LIN {X 0.380,Y -647.234,Z 1016.500,A 0.000,B 0.000,C 90.000,E1 306.011} C_DIS
LIN {X -0.177,Y -647.630,Z 1016.489,A 0.000,B 0.000,C 90.000,E1 304.072} C_DIS
LIN {X 0.005,Y -650.508,Z 1016.464,A 0.000,B 0.000,C 90.000,E1 299.589} C_DIS
LIN {X -0.254,Y -652.944,Z 1016.452,A 0.000,B 0.000,C 90.000,E1 297.385} C_DIS
LIN {X 0.174,Y -654.176,Z 1016.447,A 0.000,B 0.000,C 90.000,E1 296.360} C_DIS
LIN {X -0.255,Y -655.270,Z 1016.441,A 0.000,B 0.000,C 90.000,E1 295.412} C_DIS
LIN {X 0.200,Y -655.995,Z 1016.436,A 0.000,B 0.000,C 90.000,E1 294.387} C_DIS
LIN {X 0.160,Y -656.245,Z 1016.433,A 0.000,B 0.000,C 90.000,E1 293.898} C_DIS
LIN {X -0.360,Y -656.436,Z 1016.429,A 0.000,B 0.000,C 90.000,E1 293.206} C_DIS
LIN {X -0.166,Y -656.449,Z 1016.423,A 0.000,B 0.000,C 90.000,E1 292.206} C_DIS
LIN {X -0.194,Y -656.316,Z 1016.421,A 0.000,B 0.000,C 90.000,E1 291.716} C_DIS
LIN {X -0.219,Y -655.566,Z 1016.418,A 0.000,B 0.000,C 90.000,E1 291.227} C_DIS
LIN {X -0.116,Y -654.978,Z 1016.417,A 0.000,B 0.000,C 90.000,E1 290.972} C_DIS
LIN {X -0.248,Y -654.141,Z 1016.415,A 0.000,B 0.000,C 90.000,E1 290.737} C_DIS
LIN {X -0.151,Y -653.139,Z 1016.414,A 0.000,B 0.000,C 90.000,E1 290.482} C_DIS
LIN {X -0.104,Y -652.488,Z 1016.413,A 0.000,B 0.000,C 90.000,E1 290.355} C_DIS
LIN {X -0.240,Y -650.379,Z 1016.412,A 0.000,B 0.000,C 90.000,E1 290.120} C_DIS
LIN {X -0.158,Y -648.139,Z 1016.410,A 0.000,B 0.000,C 90.000,E1 289.866} C_DIS
LIN {X -0.338,Y -646.855,Z 1016.410,A 0.000,B 0.000,C 90.000,E1 289.758} C_DIS
LIN {X -0.259,Y -645.156,Z 1016.409,A 0.000,B 0.000,C 90.000,E1 289.631} C_DIS
LIN {X -0.094,Y -638.779,Z 1016.407,A 0.000,B 0.000,C 90.000,E1 289.214} C_DIS
LIN {X 0.123,Y -630.398,Z 1016.404,A 0.000,B 0.000,C 90.000,E1 288.779} C_DIS
LIN {X 0.192,Y -625.145,Z 1016.403,A 0.000,B 0.000,C 90.000,E1 288.544} C_DIS
LIN {X -0.211,Y -622.375,Z 1016.402,A 0.000,B 0.000,C 90.000,E1 288.417} C_DIS
LIN {X -0.244,Y -622.371,Z 1016.402,A 0.000,B 0.000,C 90.000,E1 288.417} C_DIS
LIN {X 0.112,Y -622.351,Z 1016.401,A 0.000,B 0.000,C 90.000,E1 288.236} C_DIS
LIN {X -0.063,Y -626.163,Z 1016.398,A 0.000,B 0.000,C 90.000,E1 287.692} C_DIS
LIN {X 0.295,Y -631.666,Z 1016.394,A 0.000,B 0.000,C 90.000,E1 286.913} C_DIS
LIN {X -0.268,Y -636.392,Z 1016.390,A 0.000,B 0.000,C 90.000,E1 286.205} C_DIS
LIN {X 0.003,Y -639.705,Z 1016.386,A 0.000,B 0.000,C 90.000,E1 285.552} C_DIS
LIN {X -0.320,Y -642.367,Z 1016.383,A 0.000,B 0.000,C 90.000,E1 284.954} C_DIS
LIN {X -0.009,Y -644.189,Z 1016.380,A 0.000,B 0.000,C 90.000,E1 284.426} C_DIS
LIN {X -0.001,Y -644.934,Z 1016.379,A 0.000,B 0.000,C 90.000,E1 284.175} C_DIS
LIN {X 0.328,Y -646.133,Z 1016.376,A 0.000,B 0.000,C 90.000,E1 283.647} C_DIS
LIN {X -0.103,Y -647.377,Z 1016.372,A 0.000,B 0.000,C 90.000,E1 282.939} C_DIS
LIN {X 0.247,Y -647.816,Z 1016.369,A 0.000,B 0.000,C 90.000,E1 282.411} C_DIS
LIN {X -0.168,Y -647.952,Z 1016.366,A 0.000,B 0.000,C 90.000,E1 281.951} C_DIS
LIN {X 0.190,Y -647.795,Z 1016.364,A 0.000,B 0.000,C 90.000,E1 281.422} C_DIS
LIN {X -0.234,Y -647.132,Z 1016.359,A 0.000,B 0.000,C 90.000,E1 280.715} C_DIS
LIN {X -0.004,Y -646.237,Z 1016.357,A 0.000,B 0.000,C 90.000,E1 280.197} C_DIS
LIN {X 0.335,Y -644.990,Z 1016.354,A 0.000,B 0.000,C 90.000,E1 279.670} C_DIS
LIN {X -0.077,Y -643.383,Z 1016.351,A 0.000,B 0.000,C 90.000,E1 279.208} C_DIS
LIN {X -0.235,Y -642.496,Z 1016.350,A 0.000,B 0.000,C 90.000,E1 278.973} C_DIS
LIN {X -0.025,Y -640.272,Z 1016.347,A 0.000,B 0.000,C 90.000,E1 278.454} C_DIS
LIN {X 0.124,Y -636.786,Z 1016.344,A 0.000,B 0.000,C 90.000,E1 277.814} C_DIS
LIN {X 0.293,Y -633.052,Z 1016.341,A 0.000,B 0.000,C 90.000,E1 277.296} C_DIS
LIN {X -0.189,Y -628.892,Z 1016.338,A 0.000,B 0.000,C 90.000,E1 276.834} C_DIS
LIN {X 0.076,Y -625.121,Z 1016.336,A 0.000,B 0.000,C 90.000,E1 276.429} C_DIS
LIN {X -0.214,Y -621.330,Z 1016.334,A 0.000,B 0.000,C 90.000,E1 276.087} C_DIS
LIN {X 0.276,Y -615.714,Z 1016.331,A 0.000,B 0.000,C 90.000,E1 275.568} C_DIS
LIN {X -0.253,Y -612.875,Z 1016.330,A 0.000,B 0.000,C 90.000,E1 275.391} C_DIS
LIN {X -0.007,Y -608.270,Z 1016.328,A 0.000,B 0.000,C 90.000,E1 275.049} C_DIS
LIN {X 0.129,Y -602.033,Z 1016.326,A 0.000,B 0.000,C 90.000,E1 274.645} C_DIS
LIN {X -0.065,Y -598.638,Z 1016.325,A 0.000,B 0.000,C 90.000,E1 274.473} C_DIS
LIN {X 0.055,Y -591.639,Z 1016.323,A 0.000,B 0.000,C 90.000,E1 274.131} C_DIS
LIN {X 0.242,Y -586.026,Z 1016.322,A 0.000,B 0.000,C 90.000,E1 273.898} C_DIS
LIN {X 0.214,Y -580.104,Z 1016.321,A 0.000,B 0.000,C 90.000,E1 273.726} C_DIS
LIN {X 0.094,Y -572.696,Z 1016.320,A 0.000,B 0.000,C 90.000,E1 273.555} C_DIS
LIN {X 0.095,Y -565.261,Z 1016.319,A 0.000,B 0.000,C 90.000,E1 273.440} C_DIS
LIN {X -0.233,Y -559.015,Z 1016.319,A 0.000,B 0.000,C 90.000,E1 273.440} C_DIS
LIN {X -0.255,Y -543.718,Z 1016.319,A 0.000,B 0.000,C 90.000,E1 273.440} C_DIS
LIN {X -0.055,Y -542.649,Z 1016.317,A 0.000,B 0.000,C 90.000,E1 272.980} C_DIS
LIN {X -0.241,Y -542.205,Z 1016.315,A 0.000,B 0.000,C 90.000,E1 272.694} C_DIS
LIN {X -0.027,Y -540.823,Z 1016.302,A 0.000,B 0.000,C 90.000,E1 270.401} C_DIS
LIN {X 0.061,Y -540.144,Z 1016.296,A 0.000,B 0.000,C 90.000,E1 269.255} C_DIS
LIN {X 0.169,Y -539.128,Z 1016.288,A 0.000,B 0.000,C 90.000,E1 267.822} C_DIS
LIN {X -0.229,Y -537.588,Z 1016.277,A 0.000,B 0.000,C 90.000,E1 265.869} C_DIS
LIN {X -0.089,Y -536.064,Z 1016.266,A 0.000,B 0.000,C 90.000,E1 263.856} C_DIS
LIN {X -0.016,Y -535.135,Z 1016.260,A 0.000,B 0.000,C 90.000,E1 262.704} C_DIS
LIN {X 0.157,Y -533.763,Z 1016.252,A 0.000,B 0.000,C 90.000,E1 261.254} C_DIS
LIN {X -0.216,Y -532.138,Z 1016.244,A 0.000,B 0.000,C 90.000,E1 259.859} C_DIS
LIN {X 0.082,Y -529.923,Z 1016.232,A 0.000,B 0.000,C 90.000,E1 257.813} C_DIS
LIN {X -0.264,Y -528.408,Z 1016.224,A 0.000,B 0.000,C 90.000,E1 256.408} C_DIS
LIN {X -0.031,Y -527.081,Z 1016.218,A 0.000,B 0.000,C 90.000,E1 255.227} C_DIS
LIN {X -0.172,Y -525.463,Z 1016.210,A 0.000,B 0.000,C 90.000,E1 253.795} C_DIS
LIN {X 0.159,Y -523.911,Z 1016.202,A 0.000,B 0.000,C 90.000,E1 252.308} C_DIS
LIN {X -0.031,Y -523.011,Z 1016.197,A 0.000,B 0.000,C 90.000,E1 251.456} C_DIS
LIN {X 0.059,Y -520.785,Z 1016.187,A 0.000,B 0.000,C 90.000,E1 249.699} C_DIS
LIN {X -0.066,Y -518.085,Z 1016.176,A 0.000,B 0.000,C 90.000,E1 247.667} C_DIS
LIN {X 0.145,Y -516.086,Z 1016.168,A 0.000,B 0.000,C 90.000,E1 246.177} C_DIS
LIN {X -0.065,Y -514.397,Z 1016.161,A 0.000,B 0.000,C 90.000,E1 245.025} C_DIS
LIN {X -0.167,Y -513.099,Z 1016.156,A 0.000,B 0.000,C 90.000,E1 244.152} C_DIS
LIN {X -0.077,Y -510.763,Z 1016.148,A 0.000,B 0.000,C 90.000,E1 242.666} C_DIS
LIN {X -0.064,Y -507.319,Z 1016.137,A 0.000,B 0.000,C 90.000,E1 240.589} C_DIS
LIN {X -0.159,Y -505.250,Z 1016.130,A 0.000,B 0.000,C 90.000,E1 239.410} C_DIS
LIN {X 0.091,Y -503.575,Z 1016.125,A 0.000,B 0.000,C 90.000,E1 238.486} C_DIS
LIN {X -0.063,Y -500.068,Z 1016.115,A 0.000,B 0.000,C 90.000,E1 236.707} C_DIS
LIN {X -0.157,Y -497.367,Z 1016.108,A 0.000,B 0.000,C 90.000,E1 235.515} C_DIS
LIN {X -0.146,Y -495.309,Z 1016.103,A 0.000,B 0.000,C 90.000,E1 234.609} C_DIS
LIN {X -0.163,Y -493.161,Z 1016.098,A 0.000,B 0.000,C 90.000,E1 233.703} C_DIS
LIN {X 0.151,Y -487.968,Z 1016.086,A 0.000,B 0.000,C 90.000,E1 231.537} C_DIS
LIN {X -0.075,Y -484.451,Z 1016.078,A 0.000,B 0.000,C 90.000,E1 230.033} C_DIS
LIN {X 0.049,Y -478.876,Z 1016.064,A 0.000,B 0.000,C 90.000,E1 227.553} C_DIS
LIN {X 0.037,Y -472.992,Z 1016.049,A 0.000,B 0.000,C 90.000,E1 224.757} C_DIS
LIN {X -0.005,Y -471.089,Z 1016.044,A 0.000,B 0.000,C 90.000,E1 223.824} C_DIS
LIN {X 0.169,Y -467.118,Z 1016.033,A 0.000,B 0.000,C 90.000,E1 221.919} C_DIS
LIN {X -0.185,Y -464.537,Z 1016.026,A 0.000,B 0.000,C 90.000,E1 220.701} C_DIS
LIN {X 0.071,Y -461.816,Z 1016.019,A 0.000,B 0.000,C 90.000,E1 219.402} C_DIS
LIN {X 0.084,Y -458.191,Z 1016.010,A 0.000,B 0.000,C 90.000,E1 217.810} C_DIS
LIN {X 0.122,Y -453.920,Z 1016.000,A 0.000,B 0.000,C 90.000,E1 215.884} C_DIS
LIN {X 0.002,Y -451.154,Z 1015.992,A 0.000,B 0.000,C 90.000,E1 214.612} C_DIS
LIN {X 0.051,Y -446.192,Z 1015.980,A 0.000,B 0.000,C 90.000,E1 212.339} C_DIS
LIN {X -0.128,Y -441.224,Z 1015.967,A 0.000,B 0.000,C 90.000,E1 210.079} C_DIS
LIN {X 0.050,Y -438.300,Z 1015.960,A 0.000,B 0.000,C 90.000,E1 208.743} C_DIS
LIN {X 0.005,Y -433.000,Z 1015.947,A 0.000,B 0.000,C 90.000,E1 206.437} C_DIS
LIN {X -0.167,Y -428.530,Z 1015.936,A 0.000,B 0.000,C 90.000,E1 204.463} C_DIS
LIN {X -0.137,Y -421.216,Z 1015.917,A 0.000,B 0.000,C 90.000,E1 201.099} C_DIS
LIN {X 0.095,Y -417.208,Z 1015.906,A 0.000,B 0.000,C 90.000,E1 199.033} C_DIS
LIN {X -0.151,Y -412.931,Z 1015.893,A 0.000,B 0.000,C 90.000,E1 196.677} C_DIS
LIN {X 0.158,Y -408.575,Z 1015.877,A 0.000,B 0.000,C 90.000,E1 193.883} C_DIS
LIN {X 0.049,Y -404.397,Z 1015.860,A 0.000,B 0.000,C 90.000,E1 190.782} C_DIS
LIN {X 0.134,Y -403.570,Z 1015.854,A 0.000,B 0.000,C 90.000,E1 189.726} C_DIS
LIN {X 0.135,Y -403.603,Z 1015.850,A 0.000,B 0.000,C 90.000,E1 189.029} C_DIS
LIN {X 0.074,Y -403.843,Z 1015.848,A 0.000,B 0.000,C 90.000,E1 188.690} C_DIS
LIN {X 0.079,Y -404.765,Z 1015.845,A 0.000,B 0.000,C 90.000,E1 187.992} C_DIS
LIN {X 0.083,Y -405.525,Z 1015.843,A 0.000,B 0.000,C 90.000,E1 187.644} C_DIS
LIN {X 0.089,Y -406.565,Z 1015.841,A 0.000,B 0.000,C 90.000,E1 187.296} C_DIS
LIN {X 0.113,Y -409.342,Z 1015.837,A 0.000,B 0.000,C 90.000,E1 186.606} C_DIS
LIN {X -0.131,Y -413.716,Z 1015.832,A 0.000,B 0.000,C 90.000,E1 185.853} C_DIS
LIN {X 0.072,Y -420.511,Z 1015.827,A 0.000,B 0.000,C 90.000,E1 184.878} C_DIS
LIN {X -0.142,Y -439.420,Z 1015.815,A 0.000,B 0.000,C 90.000,E1 182.636} C_DIS
LIN {X -0.207,Y -444.830,Z 1015.811,A 0.000,B 0.000,C 90.000,E1 182.007} C_DIS
LIN {X -0.009,Y -454.253,Z 1015.805,A 0.000,B 0.000,C 90.000,E1 180.859} C_DIS
LIN {X 0.131,Y -461.960,Z 1015.799,A 0.000,B 0.000,C 90.000,E1 179.885} C_DIS
LIN {X -0.007,Y -469.354,Z 1015.794,A 0.000,B 0.000,C 90.000,E1 178.969} C_DIS
LIN {X 0.147,Y -475.460,Z 1015.790,A 0.000,B 0.000,C 90.000,E1 178.165} C_DIS
LIN {X 0.154,Y -483.690,Z 1015.784,A 0.000,B 0.000,C 90.000,E1 177.078} C_DIS
LIN {X -0.030,Y -489.287,Z 1015.780,A 0.000,B 0.000,C 90.000,E1 176.331} C_DIS
LIN {X 0.004,Y -495.630,Z 1015.775,A 0.000,B 0.000,C 90.000,E1 175.412} C_DIS
LIN {X 0.156,Y -501.841,Z 1015.770,A 0.000,B 0.000,C 90.000,E1 174.489} C_DIS
LIN {X 0.118,Y -508.742,Z 1015.764,A 0.000,B 0.000,C 90.000,E1 173.457} C_DIS
LIN {X -0.237,Y -517.012,Z 1015.756,A 0.000,B 0.000,C 90.000,E1 172.186} C_DIS
LIN {X 0.167,Y -525.476,Z 1015.748,A 0.000,B 0.000,C 90.000,E1 170.679} C_DIS
LIN {X 0.127,Y -538.173,Z 1015.736,A 0.000,B 0.000,C 90.000,E1 168.522} C_DIS
LIN {X 0.170,Y -543.843,Z 1015.731,A 0.000,B 0.000,C 90.000,E1 167.521} C_DIS
LIN {X 0.161,Y -549.459,Z 1015.725,A 0.000,B 0.000,C 90.000,E1 166.533} C_DIS
LIN {X -0.210,Y -557.314,Z 1015.718,A 0.000,B 0.000,C 90.000,E1 165.172} C_DIS
LIN {X 0.216,Y -562.537,Z 1015.712,A 0.000,B 0.000,C 90.000,E1 164.157} C_DIS
LIN {X -0.098,Y -568.356,Z 1015.706,A 0.000,B 0.000,C 90.000,E1 163.087} C_DIS
LIN {X 0.190,Y -575.304,Z 1015.698,A 0.000,B 0.000,C 90.000,E1 161.692} C_DIS
LIN {X 0.224,Y -580.417,Z 1015.692,A 0.000,B 0.000,C 90.000,E1 160.604} C_DIS
LIN {X -0.155,Y -584.747,Z 1015.687,A 0.000,B 0.000,C 90.000,E1 159.699} C_DIS
LIN {X -0.222,Y -588.223,Z 1015.683,A 0.000,B 0.000,C 90.000,E1 158.901} C_DIS
LIN {X 0.179,Y -592.712,Z 1015.677,A 0.000,B 0.000,C 90.000,E1 157.794} C_DIS
LIN {X -0.362,Y -595.819,Z 1015.672,A 0.000,B 0.000,C 90.000,E1 157.050} C_DIS
LIN {X -0.169,Y -599.690,Z 1015.667,A 0.000,B 0.000,C 90.000,E1 155.973} C_DIS
LIN {X -0.098,Y -602.325,Z 1015.662,A 0.000,B 0.000,C 90.000,E1 155.177} C_DIS
LIN {X 0.186,Y -605.640,Z 1015.656,A 0.000,B 0.000,C 90.000,E1 154.101} C_DIS
LIN {X -0.076,Y -609.507,Z 1015.649,A 0.000,B 0.000,C 90.000,E1 152.820} C_DIS
LIN {X 0.081,Y -611.762,Z 1015.645,A 0.000,B 0.000,C 90.000,E1 152.025} C_DIS
LIN {X 0.186,Y -615.952,Z 1015.636,A 0.000,B 0.000,C 90.000,E1 150.461} C_DIS
LIN {X 0.135,Y -620.658,Z 1015.626,A 0.000,B 0.000,C 90.000,E1 148.663} C_DIS
LIN {X 0.191,Y -624.668,Z 1015.617,A 0.000,B 0.000,C 90.000,E1 147.120} C_DIS
LIN {X -0.206,Y -627.888,Z 1015.610,A 0.000,B 0.000,C 90.000,E1 145.881} C_DIS
LIN {X 0.171,Y -631.794,Z 1015.602,A 0.000,B 0.000,C 90.000,E1 144.322} C_DIS
LIN {X 0.259,Y -634.998,Z 1015.595,A 0.000,B 0.000,C 90.000,E1 143.050} C_DIS
LIN {X 0.002,Y -637.561,Z 1015.589,A 0.000,B 0.000,C 90.000,E1 142.065} C_DIS
LIN {X -0.036,Y -641.332,Z 1015.581,A 0.000,B 0.000,C 90.000,E1 140.561} C_DIS
LIN {X 0.177,Y -643.787,Z 1015.575,A 0.000,B 0.000,C 90.000,E1 139.542} C_DIS
LIN {X -0.076,Y -646.275,Z 1015.570,A 0.000,B 0.000,C 90.000,E1 138.566} C_DIS
LIN {X 0.227,Y -653.246,Z 1015.555,A 0.000,B 0.000,C 90.000,E1 135.810} C_DIS
LIN {X -0.143,Y -661.216,Z 1015.540,A 0.000,B 0.000,C 90.000,E1 133.137} C_DIS
LIN {X -0.201,Y -665.839,Z 1015.531,A 0.000,B 0.000,C 90.000,E1 131.676} C_DIS
LIN {X -0.168,Y -669.574,Z 1015.525,A 0.000,B 0.000,C 90.000,E1 130.458} C_DIS
LIN {X -0.087,Y -671.768,Z 1015.521,A 0.000,B 0.000,C 90.000,E1 129.725} C_DIS
LIN {X -0.388,Y -675.241,Z 1015.514,A 0.000,B 0.000,C 90.000,E1 128.543} C_DIS
LIN {X -0.101,Y -678.621,Z 1015.507,A 0.000,B 0.000,C 90.000,E1 127.317} C_DIS
LIN {X -0.147,Y -682.516,Z 1015.499,A 0.000,B 0.000,C 90.000,E1 125.884} C_DIS
LIN {X -0.145,Y -685.771,Z 1015.493,A 0.000,B 0.000,C 90.000,E1 124.692} C_DIS
LIN {X -0.097,Y -688.818,Z 1015.486,A 0.000,B 0.000,C 90.000,E1 123.499} C_DIS
LIN {X -0.161,Y -692.408,Z 1015.478,A 0.000,B 0.000,C 90.000,E1 122.084} C_DIS
LIN {X -0.043,Y -694.733,Z 1015.473,A 0.000,B 0.000,C 90.000,E1 121.131} C_DIS
LIN {X -0.255,Y -696.860,Z 1015.468,A 0.000,B 0.000,C 90.000,E1 120.207} C_DIS
LIN {X 0.252,Y -698.257,Z 1015.464,A 0.000,B 0.000,C 90.000,E1 119.461} C_DIS
LIN {X 0.012,Y -700.090,Z 1015.457,A 0.000,B 0.000,C 90.000,E1 118.309} C_DIS
LIN {X 0.209,Y -700.889,Z 1015.453,A 0.000,B 0.000,C 90.000,E1 117.590} C_DIS
LIN {X 0.227,Y -702.404,Z 1015.443,A 0.000,B 0.000,C 90.000,E1 115.720} C_DIS
LIN {X 0.129,Y -702.949,Z 1015.439,A 0.000,B 0.000,C 90.000,E1 115.027} C_DIS
LIN {X -0.242,Y -703.157,Z 1015.437,A 0.000,B 0.000,C 90.000,E1 114.591} C_DIS
LIN {X 0.319,Y -703.139,Z 1015.434,A 0.000,B 0.000,C 90.000,E1 114.079} C_DIS
LIN {X -0.051,Y -702.398,Z 1015.431,A 0.000,B 0.000,C 90.000,E1 113.643} C_DIS
LIN {X 0.226,Y -701.807,Z 1015.430,A 0.000,B 0.000,C 90.000,E1 113.387} C_DIS
LIN {X -0.149,Y -699.393,Z 1015.427,A 0.000,B 0.000,C 90.000,E1 112.950} C_DIS
LIN {X -0.017,Y -698.700,Z 1015.427,A 0.000,B 0.000,C 90.000,E1 112.823} C_DIS
LIN {X 0.116,Y -697.694,Z 1015.426,A 0.000,B 0.000,C 90.000,E1 112.695} C_DIS
LIN {X -0.024,Y -696.179,Z 1015.426,A 0.000,B 0.000,C 90.000,E1 112.589} C_DIS
LIN {X -0.148,Y -689.871,Z 1015.423,A 0.000,B 0.000,C 90.000,E1 112.206} C_DIS
LIN {X 0.139,Y -685.547,Z 1015.422,A 0.000,B 0.000,C 90.000,E1 112.025} C_DIS
LIN {X 0.000,Y -682.635,Z 1015.422,A 0.000,B 0.000,C 90.000,E1 111.972} C_DIS
LIN {X -0.263,Y -675.467,Z 1015.422,A 0.000,B 0.000,C 90.000,E1 111.897} C_DIS
LIN {X -0.292,Y -616.229,Z 1015.422,A 0.000,B 0.000,C 90.000,E1 111.897} C_DIS
LIN {X -0.202,Y -611.527,Z 1015.421,A 0.000,B 0.000,C 90.000,E1 111.770} C_DIS
LIN {X -0.270,Y -604.874,Z 1015.420,A 0.000,B 0.000,C 90.000,E1 111.535} C_DIS
LIN {X 0.250,Y -599.241,Z 1015.418,A 0.000,B 0.000,C 90.000,E1 111.227} C_DIS
LIN {X -0.204,Y -593.383,Z 1015.416,A 0.000,B 0.000,C 90.000,E1 110.918} C_DIS
LIN {X 0.072,Y -587.722,Z 1015.414,A 0.000,B 0.000,C 90.000,E1 110.482} C_DIS
LIN {X 0.037,Y -576.685,Z 1015.409,A 0.000,B 0.000,C 90.000,E1 109.577} C_DIS
LIN {X -0.052,Y -570.731,Z 1015.406,A 0.000,B 0.000,C 90.000,E1 109.141} C_DIS
LIN {X -0.108,Y -562.241,Z 1015.404,A 0.000,B 0.000,C 90.000,E1 108.671} C_DIS
LIN {X -0.231,Y -552.590,Z 1015.401,A 0.000,B 0.000,C 90.000,E1 108.181} C_DIS
LIN {X -0.095,Y -549.748,Z 1015.400,A 0.000,B 0.000,C 90.000,E1 108.000} C_DIS
LIN {X 0.140,Y -548.431,Z 1015.399,A 0.000,B 0.000,C 90.000,E1 107.819} C_DIS
LIN {X 0.099,Y -548.412,Z 1015.399,A 0.000,B 0.000,C 90.000,E1 107.819} C_DIS
LIN {X 0.055,Y -548.068,Z 1015.397,A 0.000,B 0.000,C 90.000,E1 107.402} C_DIS
LIN {X -0.008,Y -548.152,Z 1015.394,A 0.000,B 0.000,C 90.000,E1 106.858} C_DIS
LIN {X -0.101,Y -548.609,Z 1015.389,A 0.000,B 0.000,C 90.000,E1 106.024} C_DIS
LIN {X -0.171,Y -549.546,Z 1015.378,A 0.000,B 0.000,C 90.000,E1 104.064} C_DIS
LIN {X 0.214,Y -552.189,Z 1015.359,A 0.000,B 0.000,C 90.000,E1 100.658} C_DIS
LIN {X -0.097,Y -554.692,Z 1015.347,A 0.000,B 0.000,C 90.000,E1 98.454} C_DIS
LIN {X 0.075,Y -556.819,Z 1015.336,A 0.000,B 0.000,C 90.000,E1 96.486} C_DIS
LIN {X -0.028,Y -558.097,Z 1015.328,A 0.000,B 0.000,C 90.000,E1 95.106} C_DIS
LIN {X 0.249,Y -558.745,Z 1015.324,A 0.000,B 0.000,C 90.000,E1 94.245} C_DIS
LIN {X 0.179,Y -559.596,Z 1015.316,A 0.000,B 0.000,C 90.000,E1 92.865} C_DIS
LIN {X 0.179,Y -560.347,Z 1015.307,A 0.000,B 0.000,C 90.000,E1 91.203} C_DIS
LIN {X -0.277,Y -561.178,Z 1015.296,A 0.000,B 0.000,C 90.000,E1 89.312} C_DIS
LIN {X 0.126,Y -561.640,Z 1015.290,A 0.000,B 0.000,C 90.000,E1 88.165} C_DIS
LIN {X 0.079,Y -561.971,Z 1015.282,A 0.000,B 0.000,C 90.000,E1 86.788} C_DIS
LIN {X -0.213,Y -562.365,Z 1015.270,A 0.000,B 0.000,C 90.000,E1 84.609} C_DIS
LIN {X -0.165,Y -562.657,Z 1015.262,A 0.000,B 0.000,C 90.000,E1 83.223} C_DIS
LIN {X -0.122,Y -563.262,Z 1015.249,A 0.000,B 0.000,C 90.000,E1 80.735} C_DIS
LIN {X -0.040,Y -564.093,Z 1015.236,A 0.000,B 0.000,C 90.000,E1 78.522} C_DIS
LIN {X -0.157,Y -564.949,Z 1015.227,A 0.000,B 0.000,C 90.000,E1 76.881} C_DIS
LIN {X -0.195,Y -566.303,Z 1015.215,A 0.000,B 0.000,C 90.000,E1 74.685} C_DIS
LIN {X -0.307,Y -567.360,Z 1015.207,A 0.000,B 0.000,C 90.000,E1 73.323} C_DIS
LIN {X -0.247,Y -568.385,Z 1015.200,A 0.000,B 0.000,C 90.000,E1 71.945} C_DIS
LIN {X 0.007,Y -569.389,Z 1015.192,A 0.000,B 0.000,C 90.000,E1 70.550} C_DIS
LIN {X 0.130,Y -570.169,Z 1015.186,A 0.000,B 0.000,C 90.000,E1 69.444} C_DIS
LIN {X -0.121,Y -571.071,Z 1015.178,A 0.000,B 0.000,C 90.000,E1 68.103} C_DIS
LIN {X 0.033,Y -572.162,Z 1015.168,A 0.000,B 0.000,C 90.000,E1 66.177} C_DIS
LIN {X 0.084,Y -572.858,Z 1015.159,A 0.000,B 0.000,C 90.000,E1 64.537} C_DIS
LIN {X -0.110,Y -573.553,Z 1015.150,A 0.000,B 0.000,C 90.000,E1 62.922} C_DIS
LIN {X 0.218,Y -574.086,Z 1015.141,A 0.000,B 0.000,C 90.000,E1 61.257} C_DIS
LIN {X -0.018,Y -574.517,Z 1015.133,A 0.000,B 0.000,C 90.000,E1 59.921} C_DIS
LIN {X 0.254,Y -574.903,Z 1015.125,A 0.000,B 0.000,C 90.000,E1 58.535} C_DIS
LIN {X 0.314,Y -575.323,Z 1015.115,A 0.000,B 0.000,C 90.000,E1 56.628} C_DIS
LIN {X -0.218,Y -575.474,Z 1015.109,A 0.000,B 0.000,C 90.000,E1 55.595} C_DIS
LIN {X 0.200,Y -575.559,Z 1015.101,A 0.000,B 0.000,C 90.000,E1 54.196} C_DIS
LIN {X 0.151,Y -575.341,Z 1015.094,A 0.000,B 0.000,C 90.000,E1 52.844} C_DIS
LIN {X -0.059,Y -574.989,Z 1015.088,A 0.000,B 0.000,C 90.000,E1 51.778} C_DIS
LIN {X 0.076,Y -574.506,Z 1015.082,A 0.000,B 0.000,C 90.000,E1 50.678} C_DIS
LIN {X 0.275,Y -573.667,Z 1015.074,A 0.000,B 0.000,C 90.000,E1 49.299} C_DIS
LIN {X -0.044,Y -572.787,Z 1015.068,A 0.000,B 0.000,C 90.000,E1 48.243} C_DIS
LIN {X 0.301,Y -572.012,Z 1015.063,A 0.000,B 0.000,C 90.000,E1 47.391} C_DIS
LIN {X -0.172,Y -571.088,Z 1015.059,A 0.000,B 0.000,C 90.000,E1 46.620} C_DIS
LIN {X -0.261,Y -569.959,Z 1015.054,A 0.000,B 0.000,C 90.000,E1 45.810} C_DIS
LIN {X 0.045,Y -568.646,Z 1015.050,A 0.000,B 0.000,C 90.000,E1 44.960} C_DIS
LIN {X 0.334,Y -567.162,Z 1015.045,A 0.000,B 0.000,C 90.000,E1 44.109} C_DIS
LIN {X -0.111,Y -564.959,Z 1015.039,A 0.000,B 0.000,C 90.000,E1 43.056} C_DIS
LIN {X 0.239,Y -562.250,Z 1015.033,A 0.000,B 0.000,C 90.000,E1 41.919} C_DIS
LIN {X 0.006,Y -560.745,Z 1015.030,A 0.000,B 0.000,C 90.000,E1 41.391} C_DIS
LIN {X 0.130,Y -559.131,Z 1015.027,A 0.000,B 0.000,C 90.000,E1 40.825} C_DIS
LIN {X -0.044,Y -556.402,Z 1015.022,A 0.000,B 0.000,C 90.000,E1 40.011} C_DIS
LIN {X -0.171,Y -552.428,Z 1015.016,A 0.000,B 0.000,C 90.000,E1 38.910} C_DIS
LIN {X 0.022,Y -548.902,Z 1015.011,A 0.000,B 0.000,C 90.000,E1 38.051} C_DIS
LIN {X -0.300,Y -546.424,Z 1015.008,A 0.000,B 0.000,C 90.000,E1 37.523} C_DIS
LIN {X -0.144,Y -541.172,Z 1015.002,A 0.000,B 0.000,C 90.000,E1 36.377} C_DIS
LIN {X -0.079,Y -536.888,Z 1014.997,A 0.000,B 0.000,C 90.000,E1 35.518} C_DIS
LIN {X -0.069,Y -532.321,Z 1014.993,A 0.000,B 0.000,C 90.000,E1 34.659} C_DIS
LIN {X -0.132,Y -526.529,Z 1014.987,A 0.000,B 0.000,C 90.000,E1 33.658} C_DIS
LIN {X 0.195,Y -521.218,Z 1014.982,A 0.000,B 0.000,C 90.000,E1 32.752} C_DIS
LIN {X -0.195,Y -517.450,Z 1014.979,A 0.000,B 0.000,C 90.000,E1 32.212} C_DIS
LIN {X 0.005,Y -514.540,Z 1014.976,A 0.000,B 0.000,C 90.000,E1 31.750} C_DIS
LIN {X 0.095,Y -509.199,Z 1014.972,A 0.000,B 0.000,C 90.000,E1 31.003} C_DIS
LIN {X 0.063,Y -504.587,Z 1014.969,A 0.000,B 0.000,C 90.000,E1 30.413} C_DIS
LIN {X -0.056,Y -502.249,Z 1014.967,A 0.000,B 0.000,C 90.000,E1 30.129} C_DIS
LIN {X -0.290,Y -495.709,Z 1014.963,A 0.000,B 0.000,C 90.000,E1 29.411} C_DIS
LIN {X 0.240,Y -489.019,Z 1014.959,A 0.000,B 0.000,C 90.000,E1 28.615} C_DIS
LIN {X 0.193,Y -480.493,Z 1014.954,A 0.000,B 0.000,C 90.000,E1 27.769} C_DIS
LIN {X 0.104,Y -471.844,Z 1014.950,A 0.000,B 0.000,C 90.000,E1 26.950} C_DIS
LIN {X -0.045,Y -463.013,Z 1014.945,A 0.000,B 0.000,C 90.000,E1 26.155} C_DIS
LIN {X 0.260,Y -455.541,Z 1014.942,A 0.000,B 0.000,C 90.000,E1 25.463} C_DIS
LIN {X -0.041,Y -443.322,Z 1014.936,A 0.000,B 0.000,C 90.000,E1 24.463} C_DIS
LIN {X -0.128,Y -426.740,Z 1014.928,A 0.000,B 0.000,C 90.000,E1 23.003} C_DIS
LIN {X 0.027,Y -412.069,Z 1014.920,A 0.000,B 0.000,C 90.000,E1 21.535} C_DIS
LIN {X 0.046,Y -401.003,Z 1014.913,A 0.000,B 0.000,C 90.000,E1 20.301} C_DIS
LIN {X 0.057,Y -397.064,Z 1014.910,A 0.000,B 0.000,C 90.000,E1 19.812} C_DIS
LIN {X -0.139,Y -394.112,Z 1014.908,A 0.000,B 0.000,C 90.000,E1 19.396} C_DIS
LIN {X 0.077,Y -391.992,Z 1014.905,A 0.000,B 0.000,C 90.000,E1 18.906} C_DIS
LIN {X 0.173,Y -390.978,Z 1014.901,A 0.000,B 0.000,C 90.000,E1 18.236} C_DIS
LIN {X -0.215,Y -390.886,Z 1014.899,A 0.000,B 0.000,C 90.000,E1 17.764} C_DIS
LIN {X -0.036,Y -391.892,Z 1014.891,A 0.000,B 0.000,C 90.000,E1 16.315} C_DIS
LIN {X -0.054,Y -397.180,Z 1014.865,A 0.000,B 0.000,C 90.000,E1 11.715} C_DIS
LIN {X -0.163,Y -403.399,Z 1014.844,A 0.000,B 0.000,C 90.000,E1 7.871} C_DIS
LIN {X 0.141,Y -411.188,Z 1014.822,A 0.000,B 0.000,C 90.000,E1 4.012} C_DIS
LIN {X 0.151,Y -415.120,Z 1014.813,A 0.000,B 0.000,C 90.000,E1 2.293} C_DIS
LIN {X 0.181,Y -416.688,Z 1014.810,A 0.000,B 0.000,C 90.000,E1 1.776} C_DIS
LIN {X 0.057,Y -418.537,Z 1014.808,A 0.000,B 0.000,C 90.000,E1 1.375} C_DIS
LIN {X 0.035,Y -420.317,Z 1014.806,A 0.000,B 0.000,C 90.000,E1 1.088} C_DIS
LIN {X 0.063,Y -422.919,Z 1014.804,A 0.000,B 0.000,C 90.000,E1 0.745} C_DIS
LIN {X -0.135,Y -428.043,Z 1014.802,A 0.000,B 0.000,C 90.000,E1 0.344} C_DIS
LIN {X -0.212,Y -441.934,Z 1014.797,A 0.000,B 0.000,C 90.000,E1 359.542} C_DIS
LIN {X -0.071,Y -460.075,Z 1014.791,A 0.000,B 0.000,C 90.000,E1 358.453} C_DIS
LIN {X 0.044,Y -478.396,Z 1014.785,A 0.000,B 0.000,C 90.000,E1 357.364} C_DIS
LIN {X 0.062,Y -488.210,Z 1014.782,A 0.000,B 0.000,C 90.000,E1 356.788} C_DIS
LIN {X -0.073,Y -497.946,Z 1014.779,A 0.000,B 0.000,C 90.000,E1 356.216} C_DIS
LIN {X 0.237,Y -507.569,Z 1014.776,A 0.000,B 0.000,C 90.000,E1 355.584} C_DIS
LIN {X 0.155,Y -515.308,Z 1014.773,A 0.000,B 0.000,C 90.000,E1 355.065} C_DIS
LIN {X 0.037,Y -524.161,Z 1014.769,A 0.000,B 0.000,C 90.000,E1 354.432} C_DIS
LIN {X -0.093,Y -532.775,Z 1014.765,A 0.000,B 0.000,C 90.000,E1 353.742} C_DIS
LIN {X 0.020,Y -539.711,Z 1014.762,A 0.000,B 0.000,C 90.000,E1 353.109} C_DIS
LIN {X -0.110,Y -546.326,Z 1014.758,A 0.000,B 0.000,C 90.000,E1 352.470} C_DIS
LIN {X 0.190,Y -551.356,Z 1014.755,A 0.000,B 0.000,C 90.000,E1 351.894} C_DIS
LIN {X -0.215,Y -556.110,Z 1014.752,A 0.000,B 0.000,C 90.000,E1 351.376} C_DIS
LIN {X -0.203,Y -561.393,Z 1014.748,A 0.000,B 0.000,C 90.000,E1 350.679} C_DIS
LIN {X -0.145,Y -566.134,Z 1014.744,A 0.000,B 0.000,C 90.000,E1 349.982} C_DIS
LIN {X 0.199,Y -569.572,Z 1014.741,A 0.000,B 0.000,C 90.000,E1 349.398} C_DIS
LIN {X -0.156,Y -575.873,Z 1014.735,A 0.000,B 0.000,C 90.000,E1 348.342} C_DIS
LIN {X 0.031,Y -579.452,Z 1014.731,A 0.000,B 0.000,C 90.000,E1 347.645} C_DIS
LIN {X -0.195,Y -582.773,Z 1014.728,A 0.000,B 0.000,C 90.000,E1 346.992} C_DIS
LIN {X -0.052,Y -586.611,Z 1014.723,A 0.000,B 0.000,C 90.000,E1 346.172} C_DIS
LIN {X 0.219,Y -592.506,Z 1014.716,A 0.000,B 0.000,C 90.000,E1 344.810} C_DIS
LIN {X 0.311,Y -597.080,Z 1014.710,A 0.000,B 0.000,C 90.000,E1 343.740} C_DIS
LIN {X -0.113,Y -601.366,Z 1014.704,A 0.000,B 0.000,C 90.000,E1 342.725} C_DIS
LIN {X 0.276,Y -605.392,Z 1014.698,A 0.000,B 0.000,C 90.000,E1 341.638} C_DIS
LIN {X -0.082,Y -607.411,Z 1014.695,A 0.000,B 0.000,C 90.000,E1 341.148} C_DIS
LIN {X -0.180,Y -610.999,Z 1014.689,A 0.000,B 0.000,C 90.000,E1 340.115} C_DIS
LIN {X -0.233,Y -614.298,Z 1014.684,A 0.000,B 0.000,C 90.000,E1 339.082} C_DIS
LIN {X 0.007,Y -616.719,Z 1014.679,A 0.000,B 0.000,C 90.000,E1 338.284} C_DIS
LIN {X 0.239,Y -620.394,Z 1014.672,A 0.000,B 0.000,C 90.000,E1 336.975} C_DIS
LIN {X -0.034,Y -623.101,Z 1014.667,A 0.000,B 0.000,C 90.000,E1 335.973} C_DIS
LIN {X -0.275,Y -625.556,Z 1014.661,A 0.000,B 0.000,C 90.000,E1 334.973} C_DIS
LIN {X -0.199,Y -628.445,Z 1014.654,A 0.000,B 0.000,C 90.000,E1 333.691} C_DIS
LIN {X -0.127,Y -629.890,Z 1014.650,A 0.000,B 0.000,C 90.000,E1 332.922} C_DIS
LIN {X -0.012,Y -631.805,Z 1014.644,A 0.000,B 0.000,C 90.000,E1 331.897} C_DIS
LIN {X -0.090,Y -633.880,Z 1014.637,A 0.000,B 0.000,C 90.000,E1 330.639} C_DIS
LIN {X 0.061,Y -635.409,Z 1014.631,A 0.000,B 0.000,C 90.000,E1 329.616} C_DIS
LIN {X 0.365,Y -637.086,Z 1014.624,A 0.000,B 0.000,C 90.000,E1 328.329} C_DIS
LIN {X -0.218,Y -638.224,Z 1014.619,A 0.000,B 0.000,C 90.000,E1 327.375} C_DIS
LIN {X 0.137,Y -639.482,Z 1014.612,A 0.000,B 0.000,C 90.000,E1 326.087} C_DIS
LIN {X -0.060,Y -640.296,Z 1014.606,A 0.000,B 0.000,C 90.000,E1 325.102} C_DIS
LIN {X -0.242,Y -640.852,Z 1014.601,A 0.000,B 0.000,C 90.000,E1 324.116} C_DIS
LIN {X -0.016,Y -641.315,Z 1014.594,A 0.000,B 0.000,C 90.000,E1 322.844} C_DIS
LIN {X -0.299,Y -641.577,Z 1014.587,A 0.000,B 0.000,C 90.000,E1 321.618} C_DIS
LIN {X 0.136,Y -642.101,Z 1014.577,A 0.000,B 0.000,C 90.000,E1 319.828} C_DIS
LIN {X 0.020,Y -643.042,Z 1014.566,A 0.000,B 0.000,C 90.000,E1 317.838} C_DIS
LIN {X 0.114,Y -643.615,Z 1014.559,A 0.000,B 0.000,C 90.000,E1 316.581} C_DIS
LIN {X 0.002,Y -644.571,Z 1014.548,A 0.000,B 0.000,C 90.000,E1 314.595} C_DIS
LIN {X 0.119,Y -645.311,Z 1014.541,A 0.000,B 0.000,C 90.000,E1 313.338} C_DIS
LIN {X 0.181,Y -646.106,Z 1014.533,A 0.000,B 0.000,C 90.000,E1 311.838} C_DIS
LIN {X 0.235,Y -646.870,Z 1014.523,A 0.000,B 0.000,C 90.000,E1 310.092} C_DIS
LIN {X -0.115,Y -647.501,Z 1014.513,A 0.000,B 0.000,C 90.000,E1 308.382} C_DIS
LIN {X -0.298,Y -647.817,Z 1014.506,A 0.000,B 0.000,C 90.000,E1 307.156} C_DIS
LIN {X 0.046,Y -648.095,Z 1014.499,A 0.000,B 0.000,C 90.000,E1 305.884} C_DIS
LIN {X 0.354,Y -648.462,Z 1014.490,A 0.000,B 0.000,C 90.000,E1 304.119} C_DIS
LIN {X 0.237,Y -651.238,Z 1014.465,A 0.000,B 0.000,C 90.000,E1 299.667} C_DIS
LIN {X -0.096,Y -653.406,Z 1014.454,A 0.000,B 0.000,C 90.000,E1 297.719} C_DIS
LIN {X -0.019,Y -655.253,Z 1014.446,A 0.000,B 0.000,C 90.000,E1 296.232} C_DIS
LIN {X 0.160,Y -656.378,Z 1014.440,A 0.000,B 0.000,C 90.000,E1 295.232} C_DIS
LIN {X -0.083,Y -656.992,Z 1014.436,A 0.000,B 0.000,C 90.000,E1 294.515} C_DIS
LIN {X -0.116,Y -657.325,Z 1014.433,A 0.000,B 0.000,C 90.000,E1 294.027} C_DIS
LIN {X 0.237,Y -657.600,Z 1014.429,A 0.000,B 0.000,C 90.000,E1 293.259} C_DIS
LIN {X 0.194,Y -657.712,Z 1014.424,A 0.000,B 0.000,C 90.000,E1 292.280} C_DIS
LIN {X 0.178,Y -657.570,Z 1014.421,A 0.000,B 0.000,C 90.000,E1 291.791} C_DIS
LIN {X 0.290,Y -657.372,Z 1014.420,A 0.000,B 0.000,C 90.000,E1 291.535} C_DIS
LIN {X -0.340,Y -656.523,Z 1014.417,A 0.000,B 0.000,C 90.000,E1 291.099} C_DIS
LIN {X 0.378,Y -655.774,Z 1014.416,A 0.000,B 0.000,C 90.000,E1 290.791} C_DIS
LIN {X 0.250,Y -654.736,Z 1014.414,A 0.000,B 0.000,C 90.000,E1 290.556} C_DIS
LIN {X 0.349,Y -653.526,Z 1014.413,A 0.000,B 0.000,C 90.000,E1 290.301} C_DIS
LIN {X 0.170,Y -652.590,Z 1014.412,A 0.000,B 0.000,C 90.000,E1 290.194} C_DIS
LIN {X 0.260,Y -650.336,Z 1014.411,A 0.000,B 0.000,C 90.000,E1 289.939} C_DIS
LIN {X 0.302,Y -649.038,Z 1014.410,A 0.000,B 0.000,C 90.000,E1 289.812} C_DIS
LIN {X 0.261,Y -645.897,Z 1014.409,A 0.000,B 0.000,C 90.000,E1 289.577} C_DIS
LIN {X -0.090,Y -639.530,Z 1014.407,A 0.000,B 0.000,C 90.000,E1 289.214} C_DIS
LIN {X -0.006,Y -630.891,Z 1014.404,A 0.000,B 0.000,C 90.000,E1 288.779} C_DIS
LIN {X -0.136,Y -625.699,Z 1014.403,A 0.000,B 0.000,C 90.000,E1 288.544} C_DIS
LIN {X 0.135,Y -624.596,Z 1014.402,A 0.000,B 0.000,C 90.000,E1 288.417} C_DIS
LIN {X 0.079,Y -624.557,Z 1014.402,A 0.000,B 0.000,C 90.000,E1 288.417} C_DIS
LIN {X 0.273,Y -624.961,Z 1014.401,A 0.000,B 0.000,C 90.000,E1 288.236} C_DIS
LIN {X 0.236,Y -631.937,Z 1014.396,A 0.000,B 0.000,C 90.000,E1 287.221} C_DIS
LIN {X 0.041,Y -634.509,Z 1014.394,A 0.000,B 0.000,C 90.000,E1 286.858} C_DIS
LIN {X -0.317,Y -638.349,Z 1014.390,A 0.000,B 0.000,C 90.000,E1 286.260} C_DIS
LIN {X -0.033,Y -641.701,Z 1014.387,A 0.000,B 0.000,C 90.000,E1 285.607} C_DIS
LIN {X 0.286,Y -644.805,Z 1014.383,A 0.000,B 0.000,C 90.000,E1 284.828} C_DIS
LIN {X -0.012,Y -646.388,Z 1014.380,A 0.000,B 0.000,C 90.000,E1 284.356} C_DIS
LIN {X 0.190,Y -648.331,Z 1014.376,A 0.000,B 0.000,C 90.000,E1 283.592} C_DIS
LIN {X -0.084,Y -649.062,Z 1014.373,A 0.000,B 0.000,C 90.000,E1 283.119} C_DIS
LIN {X 0.146,Y -649.777,Z 1014.369,A 0.000,B 0.000,C 90.000,E1 282.355} C_DIS
LIN {X -0.122,Y -649.889,Z 1014.366,A 0.000,B 0.000,C 90.000,E1 281.883} C_DIS
LIN {X -0.016,Y -649.501,Z 1014.362,A 0.000,B 0.000,C 90.000,E1 281.130} C_DIS
LIN {X -0.289,Y -649.009,Z 1014.359,A 0.000,B 0.000,C 90.000,E1 280.658} C_DIS
LIN {X -0.044,Y -648.146,Z 1014.356,A 0.000,B 0.000,C 90.000,E1 280.141} C_DIS
LIN {X 0.310,Y -646.911,Z 1014.354,A 0.000,B 0.000,C 90.000,E1 279.613} C_DIS
LIN {X -0.090,Y -645.324,Z 1014.351,A 0.000,B 0.000,C 90.000,E1 279.151} C_DIS
LIN {X -0.242,Y -644.404,Z 1014.349,A 0.000,B 0.000,C 90.000,E1 278.916} C_DIS
LIN {X -0.017,Y -642.174,Z 1014.347,A 0.000,B 0.000,C 90.000,E1 278.398} C_DIS
LIN {X 0.281,Y -639.409,Z 1014.344,A 0.000,B 0.000,C 90.000,E1 277.871} C_DIS
LIN {X -0.299,Y -635.148,Z 1014.340,A 0.000,B 0.000,C 90.000,E1 277.296} C_DIS
LIN {X -0.276,Y -629.702,Z 1014.337,A 0.000,B 0.000,C 90.000,E1 276.663} C_DIS
LIN {X 0.004,Y -626.017,Z 1014.335,A 0.000,B 0.000,C 90.000,E1 276.258} C_DIS
LIN {X 0.288,Y -620.874,Z 1014.332,A 0.000,B 0.000,C 90.000,E1 275.739} C_DIS
LIN {X 0.221,Y -615.200,Z 1014.329,A 0.000,B 0.000,C 90.000,E1 275.277} C_DIS
LIN {X 0.263,Y -612.335,Z 1014.328,A 0.000,B 0.000,C 90.000,E1 275.049} C_DIS
LIN {X -0.231,Y -604.514,Z 1014.325,A 0.000,B 0.000,C 90.000,E1 274.588} C_DIS
LIN {X -0.153,Y -599.534,Z 1014.324,A 0.000,B 0.000,C 90.000,E1 274.302} C_DIS
LIN {X 0.011,Y -592.809,Z 1014.322,A 0.000,B 0.000,C 90.000,E1 273.955} C_DIS
LIN {X 0.042,Y -585.482,Z 1014.320,A 0.000,B 0.000,C 90.000,E1 273.669} C_DIS
LIN {X 0.095,Y -577.736,Z 1014.319,A 0.000,B 0.000,C 90.000,E1 273.440} C_DIS
LIN {X -0.092,Y -571.848,Z 1014.318,A 0.000,B 0.000,C 90.000,E1 273.326} C_DIS
LIN {X -0.051,Y -564.345,Z 1014.318,A 0.000,B 0.000,C 90.000,E1 273.212} C_DIS
LIN {X 0.187,Y -559.067,Z 1014.318,A 0.000,B 0.000,C 90.000,E1 273.154} C_DIS
LIN {X 0.144,Y -544.274,Z 1014.318,A 0.000,B 0.000,C 90.000,E1 273.154} C_DIS
LIN {X -0.153,Y -542.643,Z 1014.316,A 0.000,B 0.000,C 90.000,E1 272.808} C_DIS
LIN {X 0.059,Y -541.899,Z 1014.311,A 0.000,B 0.000,C 90.000,E1 272.007} C_DIS
LIN {X 0.224,Y -540.898,Z 1014.302,A 0.000,B 0.000,C 90.000,E1 270.286} C_DIS
LIN {X -0.207,Y -540.021,Z 1014.294,A 0.000,B 0.000,C 90.000,E1 268.912} C_DIS
LIN {X -0.119,Y -539.217,Z 1014.288,A 0.000,B 0.000,C 90.000,E1 267.764} C_DIS
LIN {X 0.023,Y -537.657,Z 1014.276,A 0.000,B 0.000,C 90.000,E1 265.755} C_DIS
LIN {X 0.160,Y -536.132,Z 1014.265,A 0.000,B 0.000,C 90.000,E1 263.742} C_DIS
LIN {X -0.252,Y -534.898,Z 1014.257,A 0.000,B 0.000,C 90.000,E1 262.356} C_DIS
LIN {X -0.128,Y -533.795,Z 1014.251,A 0.000,B 0.000,C 90.000,E1 261.197} C_DIS
LIN {X 0.023,Y -532.161,Z 1014.243,A 0.000,B 0.000,C 90.000,E1 259.746} C_DIS
LIN {X -0.205,Y -529.964,Z 1014.232,A 0.000,B 0.000,C 90.000,E1 257.757} C_DIS
LIN {X -0.039,Y -528.444,Z 1014.224,A 0.000,B 0.000,C 90.000,E1 256.297} C_DIS
LIN {X 0.166,Y -527.456,Z 1014.219,A 0.000,B 0.000,C 90.000,E1 255.408} C_DIS
LIN {X 0.030,Y -525.832,Z 1014.211,A 0.000,B 0.000,C 90.000,E1 253.976} C_DIS
LIN {X -0.134,Y -524.273,Z 1014.203,A 0.000,B 0.000,C 90.000,E1 252.543} C_DIS
LIN {X 0.169,Y -523.049,Z 1014.197,A 0.000,B 0.000,C 90.000,E1 251.348} C_DIS
LIN {X -0.059,Y -520.790,Z 1014.187,A 0.000,B 0.000,C 90.000,E1 249.625} C_DIS
LIN {X 0.307,Y -518.115,Z 1014.175,A 0.000,B 0.000,C 90.000,E1 247.539} C_DIS
LIN {X 0.046,Y -516.113,Z 1014.167,A 0.000,B 0.000,C 90.000,E1 246.102} C_DIS
LIN {X -0.253,Y -514.001,Z 1014.159,A 0.000,B 0.000,C 90.000,E1 244.665} C_DIS
LIN {X -0.029,Y -512.138,Z 1014.153,A 0.000,B 0.000,C 90.000,E1 243.461} C_DIS
LIN {X 0.038,Y -509.763,Z 1014.144,A 0.000,B 0.000,C 90.000,E1 241.975} C_DIS
LIN {X -0.137,Y -507.330,Z 1014.136,A 0.000,B 0.000,C 90.000,E1 240.511} C_DIS
LIN {X -0.228,Y -505.256,Z 1014.130,A 0.000,B 0.000,C 90.000,E1 239.331} C_DIS
LIN {X 0.023,Y -503.565,Z 1014.125,A 0.000,B 0.000,C 90.000,E1 238.408} C_DIS
LIN {X -0.001,Y -500.651,Z 1014.116,A 0.000,B 0.000,C 90.000,E1 236.914} C_DIS
LIN {X -0.086,Y -498.044,Z 1014.110,A 0.000,B 0.000,C 90.000,E1 235.722} C_DIS
LIN {X 0.200,Y -495.245,Z 1014.103,A 0.000,B 0.000,C 90.000,E1 234.482} C_DIS
LIN {X -0.218,Y -493.037,Z 1014.098,A 0.000,B 0.000,C 90.000,E1 233.623} C_DIS
LIN {X -0.046,Y -488.587,Z 1014.088,A 0.000,B 0.000,C 90.000,E1 231.778} C_DIS
LIN {X 0.242,Y -484.353,Z 1014.077,A 0.000,B 0.000,C 90.000,E1 229.908} C_DIS
LIN {X -0.127,Y -479.463,Z 1014.065,A 0.000,B 0.000,C 90.000,E1 227.796} C_DIS
LIN {X -0.222,Y -474.138,Z 1014.052,A 0.000,B 0.000,C 90.000,E1 225.324} C_DIS
LIN {X 0.262,Y -470.986,Z 1014.043,A 0.000,B 0.000,C 90.000,E1 223.704} C_DIS
LIN {X 0.178,Y -466.373,Z 1014.031,A 0.000,B 0.000,C 90.000,E1 221.515} C_DIS
LIN {X 0.161,Y -463.715,Z 1014.024,A 0.000,B 0.000,C 90.000,E1 220.253} C_DIS
LIN {X 0.110,Y -460.941,Z 1014.017,A 0.000,B 0.000,C 90.000,E1 218.991} C_DIS
LIN {X -0.143,Y -455.899,Z 1014.004,A 0.000,B 0.000,C 90.000,E1 216.790} C_DIS
LIN {X 0.206,Y -451.740,Z 1013.994,A 0.000,B 0.000,C 90.000,E1 214.818} C_DIS
LIN {X -0.040,Y -446.021,Z 1013.979,A 0.000,B 0.000,C 90.000,E1 212.260} C_DIS
LIN {X -0.280,Y -441.759,Z 1013.968,A 0.000,B 0.000,C 90.000,E1 210.335} C_DIS
LIN {X -0.092,Y -438.854,Z 1013.961,A 0.000,B 0.000,C 90.000,E1 208.999} C_DIS
LIN {X 0.214,Y -435.834,Z 1013.954,A 0.000,B 0.000,C 90.000,E1 207.641} C_DIS
LIN {X 0.098,Y -430.607,Z 1013.941,A 0.000,B 0.000,C 90.000,E1 205.335} C_DIS
LIN {X -0.097,Y -427.564,Z 1013.933,A 0.000,B 0.000,C 90.000,E1 204.027} C_DIS
LIN {X 0.111,Y -421.020,Z 1013.917,A 0.000,B 0.000,C 90.000,E1 200.972} C_DIS
LIN {X -0.062,Y -416.986,Z 1013.905,A 0.000,B 0.000,C 90.000,E1 198.960} C_DIS
LIN {X 0.073,Y -412.685,Z 1013.892,A 0.000,B 0.000,C 90.000,E1 196.551} C_DIS
LIN {X -0.148,Y -408.826,Z 1013.879,A 0.000,B 0.000,C 90.000,E1 194.175} C_DIS
LIN {X 0.139,Y -404.895,Z 1013.863,A 0.000,B 0.000,C 90.000,E1 191.366} C_DIS
LIN {X -0.162,Y -403.371,Z 1013.856,A 0.000,B 0.000,C 90.000,E1 190.018} C_DIS
LIN {X -0.162,Y -403.122,Z 1013.854,A 0.000,B 0.000,C 90.000,E1 189.670} C_DIS
LIN {X -0.163,Y -402.962,Z 1013.850,A 0.000,B 0.000,C 90.000,E1 188.973} C_DIS
LIN {X -0.165,Y -403.225,Z 1013.848,A 0.000,B 0.000,C 90.000,E1 188.624} C_DIS
LIN {X -0.170,Y -404.104,Z 1013.844,A 0.000,B 0.000,C 90.000,E1 187.928} C_DIS
LIN {X 0.203,Y -404.197,Z 1013.843,A 0.000,B 0.000,C 90.000,E1 187.701} C_DIS
LIN {X 0.087,Y -404.960,Z 1013.841,A 0.000,B 0.000,C 90.000,E1 187.352} C_DIS
LIN {X 0.090,Y -406.000,Z 1013.839,A 0.000,B 0.000,C 90.000,E1 187.004} C_DIS
LIN {X 0.043,Y -408.560,Z 1013.836,A 0.000,B 0.000,C 90.000,E1 186.372} C_DIS
LIN {X 0.014,Y -410.372,Z 1013.834,A 0.000,B 0.000,C 90.000,E1 186.030} C_DIS
LIN {X 0.029,Y -413.367,Z 1013.831,A 0.000,B 0.000,C 90.000,E1 185.511} C_DIS
LIN {X -0.172,Y -418.934,Z 1013.826,A 0.000,B 0.000,C 90.000,E1 184.759} C_DIS
LIN {X 0.174,Y -435.365,Z 1013.815,A 0.000,B 0.000,C 90.000,E1 182.751} C_DIS
LIN {X 0.059,Y -443.426,Z 1013.810,A 0.000,B 0.000,C 90.000,E1 181.835} C_DIS
LIN {X -0.095,Y -454.197,Z 1013.803,A 0.000,B 0.000,C 90.000,E1 180.573} C_DIS
LIN {X 0.161,Y -463.239,Z 1013.797,A 0.000,B 0.000,C 90.000,E1 179.427} C_DIS
LIN {X 0.134,Y -468.381,Z 1013.793,A 0.000,B 0.000,C 90.000,E1 178.797} C_DIS
LIN {X -0.062,Y -475.770,Z 1013.788,A 0.000,B 0.000,C 90.000,E1 177.879} C_DIS
LIN {X 0.136,Y -481.771,Z 1013.784,A 0.000,B 0.000,C 90.000,E1 177.078} C_DIS
LIN {X 0.087,Y -488.618,Z 1013.779,A 0.000,B 0.000,C 90.000,E1 176.159} C_DIS
LIN {X 0.002,Y -497.111,Z 1013.772,A 0.000,B 0.000,C 90.000,E1 174.951} C_DIS
LIN {X 0.123,Y -503.261,Z 1013.767,A 0.000,B 0.000,C 90.000,E1 174.033} C_DIS
LIN {X 0.055,Y -510.087,Z 1013.761,A 0.000,B 0.000,C 90.000,E1 172.996} C_DIS
LIN {X -0.088,Y -517.516,Z 1013.755,A 0.000,B 0.000,C 90.000,E1 171.837} C_DIS
LIN {X 0.195,Y -526.815,Z 1013.746,A 0.000,B 0.000,C 90.000,E1 170.208} C_DIS
LIN {X 0.143,Y -537.900,Z 1013.735,A 0.000,B 0.000,C 90.000,E1 168.342} C_DIS
LIN {X -0.297,Y -546.885,Z 1013.727,A 0.000,B 0.000,C 90.000,E1 166.825} C_DIS
LIN {X -0.197,Y -557.147,Z 1013.717,A 0.000,B 0.000,C 90.000,E1 164.991} C_DIS
LIN {X -0.047,Y -563.065,Z 1013.710,A 0.000,B 0.000,C 90.000,E1 163.866} C_DIS
LIN {X -0.087,Y -568.122,Z 1013.705,A 0.000,B 0.000,C 90.000,E1 162.906} C_DIS
LIN {X 0.292,Y -574.413,Z 1013.698,A 0.000,B 0.000,C 90.000,E1 161.638} C_DIS
LIN {X -0.154,Y -578.939,Z 1013.693,A 0.000,B 0.000,C 90.000,E1 160.732} C_DIS
LIN {X -0.081,Y -583.932,Z 1013.687,A 0.000,B 0.000,C 90.000,E1 159.645} C_DIS
LIN {X -0.158,Y -587.489,Z 1013.682,A 0.000,B 0.000,C 90.000,E1 158.847} C_DIS
LIN {X -0.319,Y -592.003,Z 1013.677,A 0.000,B 0.000,C 90.000,E1 157.794} C_DIS
LIN {X -0.087,Y -595.120,Z 1013.672,A 0.000,B 0.000,C 90.000,E1 156.975} C_DIS
LIN {X -0.141,Y -599.060,Z 1013.666,A 0.000,B 0.000,C 90.000,E1 155.921} C_DIS
LIN {X 0.102,Y -602.616,Z 1013.660,A 0.000,B 0.000,C 90.000,E1 154.845} C_DIS
LIN {X -0.146,Y -605.880,Z 1013.655,A 0.000,B 0.000,C 90.000,E1 153.819} C_DIS
LIN {X 0.145,Y -609.705,Z 1013.647,A 0.000,B 0.000,C 90.000,E1 152.487} C_DIS
LIN {X 0.275,Y -612.581,Z 1013.641,A 0.000,B 0.000,C 90.000,E1 151.435} C_DIS
LIN {X 0.147,Y -615.435,Z 1013.636,A 0.000,B 0.000,C 90.000,E1 150.411} C_DIS
LIN {X 0.072,Y -620.192,Z 1013.626,A 0.000,B 0.000,C 90.000,E1 148.614} C_DIS
LIN {X -0.076,Y -624.210,Z 1013.617,A 0.000,B 0.000,C 90.000,E1 147.089} C_DIS
LIN {X 0.041,Y -628.129,Z 1013.609,A 0.000,B 0.000,C 90.000,E1 145.548} C_DIS
LIN {X -0.093,Y -632.065,Z 1013.600,A 0.000,B 0.000,C 90.000,E1 144.036} C_DIS
LIN {X 0.377,Y -635.958,Z 1013.592,A 0.000,B 0.000,C 90.000,E1 142.477} C_DIS
LIN {X -0.087,Y -639.788,Z 1013.583,A 0.000,B 0.000,C 90.000,E1 141.009} C_DIS
LIN {X -0.068,Y -643.505,Z 1013.575,A 0.000,B 0.000,C 90.000,E1 139.504} C_DIS
LIN {X 0.167,Y -645.994,Z 1013.570,A 0.000,B 0.000,C 90.000,E1 138.485} C_DIS
LIN {X 0.373,Y -648.433,Z 1013.564,A 0.000,B 0.000,C 90.000,E1 137.472} C_DIS
LIN {X -0.037,Y -653.754,Z 1013.553,A 0.000,B 0.000,C 90.000,E1 135.526} C_DIS
LIN {X 0.092,Y -661.115,Z 1013.539,A 0.000,B 0.000,C 90.000,E1 133.056} C_DIS
LIN {X 0.022,Y -666.560,Z 1013.530,A 0.000,B 0.000,C 90.000,E1 131.353} C_DIS
LIN {X 0.144,Y -671.062,Z 1013.522,A 0.000,B 0.000,C 90.000,E1 129.886} C_DIS
LIN {X -0.156,Y -675.251,Z 1013.514,A 0.000,B 0.000,C 90.000,E1 128.463} C_DIS
LIN {X 0.129,Y -678.644,Z 1013.507,A 0.000,B 0.000,C 90.000,E1 127.237} C_DIS
LIN {X 0.081,Y -682.559,Z 1013.499,A 0.000,B 0.000,C 90.000,E1 125.804} C_DIS
LIN {X 0.083,Y -685.804,Z 1013.492,A 0.000,B 0.000,C 90.000,E1 124.612} C_DIS
LIN {X 0.129,Y -688.873,Z 1013.486,A 0.000,B 0.000,C 90.000,E1 123.420} C_DIS
LIN {X 0.061,Y -692.444,Z 1013.478,A 0.000,B 0.000,C 90.000,E1 122.005} C_DIS
LIN {X 0.177,Y -694.775,Z 1013.473,A 0.000,B 0.000,C 90.000,E1 121.052} C_DIS
LIN {X -0.038,Y -696.896,Z 1013.467,A 0.000,B 0.000,C 90.000,E1 120.129} C_DIS
LIN {X 0.123,Y -698.277,Z 1013.464,A 0.000,B 0.000,C 90.000,E1 119.411} C_DIS
LIN {X 0.222,Y -700.135,Z 1013.457,A 0.000,B 0.000,C 90.000,E1 118.231} C_DIS
LIN {X 0.416,Y -700.870,Z 1013.453,A 0.000,B 0.000,C 90.000,E1 117.513} C_DIS
LIN {X 0.119,Y -702.397,Z 1013.443,A 0.000,B 0.000,C 90.000,E1 115.668} C_DIS
LIN {X -0.333,Y -703.055,Z 1013.438,A 0.000,B 0.000,C 90.000,E1 114.771} C_DIS
LIN {X 0.226,Y -703.116,Z 1013.435,A 0.000,B 0.000,C 90.000,E1 114.259} C_DIS
LIN {X 0.218,Y -702.984,Z 1013.434,A 0.000,B 0.000,C 90.000,E1 114.027} C_DIS
LIN {X 0.132,Y -702.244,Z 1013.431,A 0.000,B 0.000,C 90.000,E1 113.567} C_DIS
LIN {X 0.128,Y -701.442,Z 1013.430,A 0.000,B 0.000,C 90.000,E1 113.334} C_DIS
LIN {X -0.247,Y -699.059,Z 1013.427,A 0.000,B 0.000,C 90.000,E1 112.898} C_DIS
LIN {X -0.114,Y -698.226,Z 1013.427,A 0.000,B 0.000,C 90.000,E1 112.770} C_DIS
LIN {X 0.018,Y -696.990,Z 1013.426,A 0.000,B 0.000,C 90.000,E1 112.642} C_DIS
LIN {X 0.289,Y -690.589,Z 1013.424,A 0.000,B 0.000,C 90.000,E1 112.206} C_DIS
LIN {X -0.200,Y -688.647,Z 1013.423,A 0.000,B 0.000,C 90.000,E1 112.153} C_DIS
LIN {X 0.208,Y -685.839,Z 1013.422,A 0.000,B 0.000,C 90.000,E1 112.025} C_DIS
LIN {X 0.160,Y -683.816,Z 1013.422,A 0.000,B 0.000,C 90.000,E1 111.972} C_DIS
LIN {X -0.311,Y -675.531,Z 1013.422,A 0.000,B 0.000,C 90.000,E1 111.897} C_DIS
LIN {X 0.278,Y -674.989,Z 1013.422,A 0.000,B 0.000,C 90.000,E1 111.844} C_DIS
LIN {X 0.218,Y -616.593,Z 1013.422,A 0.000,B 0.000,C 90.000,E1 111.844} C_DIS
LIN {X 0.201,Y -611.572,Z 1013.421,A 0.000,B 0.000,C 90.000,E1 111.716} C_DIS
LIN {X 0.111,Y -604.923,Z 1013.419,A 0.000,B 0.000,C 90.000,E1 111.482} C_DIS
LIN {X 0.078,Y -599.265,Z 1013.418,A 0.000,B 0.000,C 90.000,E1 111.227} C_DIS
LIN {X 0.180,Y -593.399,Z 1013.416,A 0.000,B 0.000,C 90.000,E1 110.865} C_DIS
LIN {X -0.077,Y -587.755,Z 1013.414,A 0.000,B 0.000,C 90.000,E1 110.482} C_DIS
LIN {X -0.080,Y -578.114,Z 1013.409,A 0.000,B 0.000,C 90.000,E1 109.685} C_DIS
LIN {X 0.055,Y -572.174,Z 1013.407,A 0.000,B 0.000,C 90.000,E1 109.214} C_DIS
LIN {X 0.207,Y -570.485,Z 1013.406,A 0.000,B 0.000,C 90.000,E1 109.087} C_DIS
LIN {X 0.036,Y -563.859,Z 1013.404,A 0.000,B 0.000,C 90.000,E1 108.725} C_DIS
LIN {X -0.286,Y -552.690,Z 1013.401,A 0.000,B 0.000,C 90.000,E1 108.181} C_DIS
LIN {X -0.244,Y -549.669,Z 1013.400,A 0.000,B 0.000,C 90.000,E1 108.000} C_DIS
LIN {X 0.145,Y -548.487,Z 1013.399,A 0.000,B 0.000,C 90.000,E1 107.819} C_DIS
LIN {X 0.103,Y -548.454,Z 1013.399,A 0.000,B 0.000,C 90.000,E1 107.819} C_DIS
LIN {X -0.109,Y -548.107,Z 1013.397,A 0.000,B 0.000,C 90.000,E1 107.402} C_DIS
LIN {X -0.172,Y -548.192,Z 1013.394,A 0.000,B 0.000,C 90.000,E1 106.858} C_DIS
LIN {X 0.168,Y -548.563,Z 1013.391,A 0.000,B 0.000,C 90.000,E1 106.260} C_DIS
LIN {X 0.199,Y -549.590,Z 1013.378,A 0.000,B 0.000,C 90.000,E1 104.008} C_DIS
LIN {X 0.051,Y -552.236,Z 1013.359,A 0.000,B 0.000,C 90.000,E1 100.658} C_DIS
LIN {X -0.259,Y -554.743,Z 1013.347,A 0.000,B 0.000,C 90.000,E1 98.454} C_DIS
LIN {X -0.085,Y -556.864,Z 1013.336,A 0.000,B 0.000,C 90.000,E1 96.486} C_DIS
LIN {X -0.189,Y -558.110,Z 1013.328,A 0.000,B 0.000,C 90.000,E1 95.106} C_DIS
LIN {X 0.089,Y -558.755,Z 1013.324,A 0.000,B 0.000,C 90.000,E1 94.245} C_DIS
LIN {X 0.019,Y -559.606,Z 1013.316,A 0.000,B 0.000,C 90.000,E1 92.865} C_DIS
LIN {X 0.019,Y -560.354,Z 1013.307,A 0.000,B 0.000,C 90.000,E1 91.203} C_DIS
LIN {X 0.124,Y -561.217,Z 1013.296,A 0.000,B 0.000,C 90.000,E1 89.255} C_DIS
LIN {X -0.034,Y -561.674,Z 1013.290,A 0.000,B 0.000,C 90.000,E1 88.165} C_DIS
LIN {X -0.081,Y -562.001,Z 1013.282,A 0.000,B 0.000,C 90.000,E1 86.788} C_DIS
LIN {X -0.231,Y -562.419,Z 1013.268,A 0.000,B 0.000,C 90.000,E1 84.318} C_DIS
LIN {X 0.234,Y -562.650,Z 1013.262,A 0.000,B 0.000,C 90.000,E1 83.166} C_DIS
LIN {X 0.060,Y -562.740,Z 1013.258,A 0.000,B 0.000,C 90.000,E1 82.356} C_DIS
LIN {X 0.115,Y -563.142,Z 1013.250,A 0.000,B 0.000,C 90.000,E1 80.971} C_DIS
LIN {X -0.202,Y -564.099,Z 1013.236,A 0.000,B 0.000,C 90.000,E1 78.522} C_DIS
LIN {X -0.154,Y -565.085,Z 1013.225,A 0.000,B 0.000,C 90.000,E1 76.589} C_DIS
LIN {X 0.291,Y -566.969,Z 1013.210,A 0.000,B 0.000,C 90.000,E1 73.795} C_DIS
LIN {X -0.029,Y -568.173,Z 1013.201,A 0.000,B 0.000,C 90.000,E1 72.181} C_DIS
LIN {X -0.117,Y -568.988,Z 1013.195,A 0.000,B 0.000,C 90.000,E1 71.094} C_DIS
LIN {X 0.151,Y -569.963,Z 1013.187,A 0.000,B 0.000,C 90.000,E1 69.699} C_DIS
LIN {X -0.286,Y -571.027,Z 1013.178,A 0.000,B 0.000,C 90.000,E1 68.103} C_DIS
LIN {X -0.133,Y -572.114,Z 1013.168,A 0.000,B 0.000,C 90.000,E1 66.177} C_DIS
LIN {X -0.083,Y -572.799,Z 1013.159,A 0.000,B 0.000,C 90.000,E1 64.537} C_DIS
LIN {X 0.231,Y -573.472,Z 1013.149,A 0.000,B 0.000,C 90.000,E1 62.871} C_DIS
LIN {X 0.046,Y -573.961,Z 1013.140,A 0.000,B 0.000,C 90.000,E1 61.257} C_DIS
LIN {X -0.192,Y -574.393,Z 1013.133,A 0.000,B 0.000,C 90.000,E1 59.921} C_DIS
LIN {X 0.077,Y -574.783,Z 1013.125,A 0.000,B 0.000,C 90.000,E1 58.535} C_DIS
LIN {X 0.134,Y -575.176,Z 1013.115,A 0.000,B 0.000,C 90.000,E1 56.628} C_DIS
LIN {X 0.075,Y -575.325,Z 1013.109,A 0.000,B 0.000,C 90.000,E1 55.548} C_DIS
LIN {X 0.017,Y -575.384,Z 1013.101,A 0.000,B 0.000,C 90.000,E1 54.196} C_DIS
LIN {X -0.036,Y -575.160,Z 1013.094,A 0.000,B 0.000,C 90.000,E1 52.844} C_DIS
LIN {X 0.108,Y -574.787,Z 1013.088,A 0.000,B 0.000,C 90.000,E1 51.743} C_DIS
LIN {X 0.249,Y -574.288,Z 1013.082,A 0.000,B 0.000,C 90.000,E1 50.642} C_DIS
LIN {X 0.080,Y -573.443,Z 1013.074,A 0.000,B 0.000,C 90.000,E1 49.299} C_DIS
LIN {X -0.242,Y -572.536,Z 1013.068,A 0.000,B 0.000,C 90.000,E1 48.243} C_DIS
LIN {X 0.100,Y -571.730,Z 1013.063,A 0.000,B 0.000,C 90.000,E1 47.391} C_DIS
LIN {X 0.017,Y -570.792,Z 1013.059,A 0.000,B 0.000,C 90.000,E1 46.581} C_DIS
LIN {X -0.166,Y -570.091,Z 1013.056,A 0.000,B 0.000,C 90.000,E1 46.053} C_DIS
LIN {X 0.238,Y -568.272,Z 1013.050,A 0.000,B 0.000,C 90.000,E1 44.919} C_DIS
LIN {X 0.123,Y -566.775,Z 1013.045,A 0.000,B 0.000,C 90.000,E1 44.109} C_DIS
LIN {X 0.085,Y -564.536,Z 1013.039,A 0.000,B 0.000,C 90.000,E1 43.014} C_DIS
LIN {X 0.017,Y -561.761,Z 1013.033,A 0.000,B 0.000,C 90.000,E1 41.919} C_DIS
LIN {X -0.219,Y -560.229,Z 1013.030,A 0.000,B 0.000,C 90.000,E1 41.391} C_DIS
LIN {X -0.097,Y -558.563,Z 1013.027,A 0.000,B 0.000,C 90.000,E1 40.825} C_DIS
LIN {X -0.277,Y -555.791,Z 1013.022,A 0.000,B 0.000,C 90.000,E1 40.011} C_DIS
LIN {X 0.298,Y -552.771,Z 1013.018,A 0.000,B 0.000,C 90.000,E1 39.116} C_DIS
LIN {X -0.064,Y -551.726,Z 1013.016,A 0.000,B 0.000,C 90.000,E1 38.874} C_DIS
LIN {X 0.116,Y -548.155,Z 1013.011,A 0.000,B 0.000,C 90.000,E1 38.016} C_DIS
LIN {X 0.256,Y -544.335,Z 1013.007,A 0.000,B 0.000,C 90.000,E1 37.156} C_DIS
LIN {X 0.204,Y -539.596,Z 1013.001,A 0.000,B 0.000,C 90.000,E1 36.171} C_DIS
LIN {X 0.248,Y -535.262,Z 1012.996,A 0.000,B 0.000,C 90.000,E1 35.311} C_DIS
LIN {X -0.063,Y -530.539,Z 1012.992,A 0.000,B 0.000,C 90.000,E1 34.485} C_DIS
LIN {X 0.152,Y -524.679,Z 1012.986,A 0.000,B 0.000,C 90.000,E1 33.452} C_DIS
LIN {X -0.098,Y -520.160,Z 1012.982,A 0.000,B 0.000,C 90.000,E1 32.752} C_DIS
LIN {X 0.220,Y -516.328,Z 1012.979,A 0.000,B 0.000,C 90.000,E1 32.133} C_DIS
LIN {X -0.027,Y -513.341,Z 1012.976,A 0.000,B 0.000,C 90.000,E1 31.720} C_DIS
LIN {X -0.033,Y -509.066,Z 1012.973,A 0.000,B 0.000,C 90.000,E1 31.131} C_DIS
LIN {X 0.001,Y -503.232,Z 1012.969,A 0.000,B 0.000,C 90.000,E1 30.384} C_DIS
LIN {X 0.119,Y -499.484,Z 1012.966,A 0.000,B 0.000,C 90.000,E1 29.922} C_DIS
LIN {X -0.082,Y -492.952,Z 1012.962,A 0.000,B 0.000,C 90.000,E1 29.205} C_DIS
LIN {X 0.074,Y -488.847,Z 1012.960,A 0.000,B 0.000,C 90.000,E1 28.743} C_DIS
LIN {X 0.037,Y -480.325,Z 1012.955,A 0.000,B 0.000,C 90.000,E1 27.897} C_DIS
LIN {X 0.038,Y -473.146,Z 1012.951,A 0.000,B 0.000,C 90.000,E1 27.206} C_DIS
LIN {X -0.056,Y -464.469,Z 1012.947,A 0.000,B 0.000,C 90.000,E1 26.411} C_DIS
LIN {X 0.254,Y -457.071,Z 1012.943,A 0.000,B 0.000,C 90.000,E1 25.720} C_DIS
LIN {X -0.045,Y -444.861,Z 1012.937,A 0.000,B 0.000,C 90.000,E1 24.719} C_DIS
LIN {X 0.131,Y -425.159,Z 1012.928,A 0.000,B 0.000,C 90.000,E1 22.950} C_DIS
LIN {X 0.100,Y -409.738,Z 1012.919,A 0.000,B 0.000,C 90.000,E1 21.408} C_DIS
LIN {X 0.067,Y -398.848,Z 1012.912,A 0.000,B 0.000,C 90.000,E1 20.174} C_DIS
LIN {X -0.009,Y -396.511,Z 1012.911,A 0.000,B 0.000,C 90.000,E1 19.885} C_DIS
LIN {X -0.046,Y -394.825,Z 1012.909,A 0.000,B 0.000,C 90.000,E1 19.631} C_DIS
LIN {X 0.036,Y -393.150,Z 1012.907,A 0.000,B 0.000,C 90.000,E1 19.322} C_DIS
LIN {X -0.148,Y -391.947,Z 1012.906,A 0.000,B 0.000,C 90.000,E1 19.033} C_DIS
LIN {X -0.005,Y -391.551,Z 1012.905,A 0.000,B 0.000,C 90.000,E1 18.852} C_DIS
LIN {X -0.185,Y -390.871,Z 1012.902,A 0.000,B 0.000,C 90.000,E1 18.362} C_DIS
LIN {X -0.094,Y -390.910,Z 1012.898,A 0.000,B 0.000,C 90.000,E1 17.638} C_DIS
LIN {X 0.041,Y -396.453,Z 1012.868,A 0.000,B 0.000,C 90.000,E1 12.299} C_DIS
LIN {X -0.103,Y -403.047,Z 1012.845,A 0.000,B 0.000,C 90.000,E1 8.106} C_DIS
LIN {X -0.178,Y -408.464,Z 1012.830,A 0.000,B 0.000,C 90.000,E1 5.334} C_DIS
LIN {X -0.188,Y -413.790,Z 1012.816,A 0.000,B 0.000,C 90.000,E1 2.922} C_DIS
LIN {X -0.180,Y -415.442,Z 1012.812,A 0.000,B 0.000,C 90.000,E1 2.236} C_DIS
LIN {X -0.150,Y -417.015,Z 1012.810,A 0.000,B 0.000,C 90.000,E1 1.718} C_DIS
LIN {X -0.019,Y -419.633,Z 1012.806,A 0.000,B 0.000,C 90.000,E1 1.146} C_DIS
LIN {X -0.007,Y -420.738,Z 1012.805,A 0.000,B 0.000,C 90.000,E1 0.974} C_DIS
LIN {X 0.000,Y -423.557,Z 1012.804,A 0.000,B 0.000,C 90.000,E1 0.630} C_DIS
LIN {X -0.110,Y -427.147,Z 1012.802,A 0.000,B 0.000,C 90.000,E1 0.344} C_DIS
LIN {X 0.190,Y -429.028,Z 1012.801,A 0.000,B 0.000,C 90.000,E1 0.172} C_DIS
LIN {X -0.029,Y -442.388,Z 1012.797,A 0.000,B 0.000,C 90.000,E1 359.427} C_DIS
LIN {X 0.152,Y -460.516,Z 1012.791,A 0.000,B 0.000,C 90.000,E1 358.339} C_DIS
LIN {X 0.019,Y -480.437,Z 1012.784,A 0.000,B 0.000,C 90.000,E1 357.192} C_DIS
LIN {X -0.150,Y -488.637,Z 1012.782,A 0.000,B 0.000,C 90.000,E1 356.731} C_DIS
LIN {X -0.057,Y -501.730,Z 1012.777,A 0.000,B 0.000,C 90.000,E1 355.927} C_DIS
LIN {X -0.037,Y -508.107,Z 1012.775,A 0.000,B 0.000,C 90.000,E1 355.527} C_DIS
LIN {X -0.149,Y -515.977,Z 1012.772,A 0.000,B 0.000,C 90.000,E1 355.008} C_DIS
LIN {X 0.050,Y -524.971,Z 1012.768,A 0.000,B 0.000,C 90.000,E1 354.318} C_DIS
LIN {X 0.090,Y -532.038,Z 1012.765,A 0.000,B 0.000,C 90.000,E1 353.742} C_DIS
LIN {X 0.247,Y -538.998,Z 1012.762,A 0.000,B 0.000,C 90.000,E1 353.109} C_DIS
LIN {X 0.164,Y -545.638,Z 1012.758,A 0.000,B 0.000,C 90.000,E1 352.470} C_DIS
LIN {X -0.026,Y -550.778,Z 1012.755,A 0.000,B 0.000,C 90.000,E1 351.951} C_DIS
LIN {X 0.170,Y -555.530,Z 1012.752,A 0.000,B 0.000,C 90.000,E1 351.376} C_DIS
LIN {X 0.180,Y -560.923,Z 1012.748,A 0.000,B 0.000,C 90.000,E1 350.679} C_DIS
LIN {X -0.072,Y -564.862,Z 1012.745,A 0.000,B 0.000,C 90.000,E1 350.151} C_DIS
LIN {X 0.021,Y -569.267,Z 1012.741,A 0.000,B 0.000,C 90.000,E1 349.454} C_DIS
LIN {X 0.226,Y -575.609,Z 1012.735,A 0.000,B 0.000,C 90.000,E1 348.342} C_DIS
LIN {X -0.154,Y -579.249,Z 1012.732,A 0.000,B 0.000,C 90.000,E1 347.701} C_DIS
LIN {X 0.186,Y -582.589,Z 1012.728,A 0.000,B 0.000,C 90.000,E1 346.992} C_DIS
LIN {X 0.007,Y -587.686,Z 1012.722,A 0.000,B 0.000,C 90.000,E1 345.936} C_DIS
LIN {X 0.297,Y -593.598,Z 1012.715,A 0.000,B 0.000,C 90.000,E1 344.574} C_DIS
LIN {X -0.171,Y -598.121,Z 1012.709,A 0.000,B 0.000,C 90.000,E1 343.559} C_DIS
LIN {X -0.009,Y -602.389,Z 1012.703,A 0.000,B 0.000,C 90.000,E1 342.489} C_DIS
LIN {X 0.116,Y -607.419,Z 1012.695,A 0.000,B 0.000,C 90.000,E1 341.167} C_DIS
LIN {X 0.217,Y -611.099,Z 1012.690,A 0.000,B 0.000,C 90.000,E1 340.115} C_DIS
LIN {X 0.167,Y -614.411,Z 1012.684,A 0.000,B 0.000,C 90.000,E1 339.082} C_DIS
LIN {X -0.163,Y -616.844,Z 1012.680,A 0.000,B 0.000,C 90.000,E1 338.337} C_DIS
LIN {X -0.168,Y -620.567,Z 1012.672,A 0.000,B 0.000,C 90.000,E1 337.050} C_DIS
LIN {X 0.125,Y -623.291,Z 1012.667,A 0.000,B 0.000,C 90.000,E1 335.997} C_DIS
LIN {X 0.141,Y -625.777,Z 1012.661,A 0.000,B 0.000,C 90.000,E1 334.973} C_DIS
LIN {X -0.056,Y -628.691,Z 1012.654,A 0.000,B 0.000,C 90.000,E1 333.717} C_DIS
LIN {X 0.011,Y -630.180,Z 1012.650,A 0.000,B 0.000,C 90.000,E1 332.948} C_DIS
LIN {X -0.140,Y -632.106,Z 1012.644,A 0.000,B 0.000,C 90.000,E1 331.948} C_DIS
LIN {X 0.072,Y -634.626,Z 1012.636,A 0.000,B 0.000,C 90.000,E1 330.411} C_DIS
LIN {X -0.006,Y -636.137,Z 1012.630,A 0.000,B 0.000,C 90.000,E1 329.410} C_DIS
LIN {X 0.313,Y -637.788,Z 1012.623,A 0.000,B 0.000,C 90.000,E1 328.122} C_DIS
LIN {X 0.278,Y -638.922,Z 1012.617,A 0.000,B 0.000,C 90.000,E1 327.120} C_DIS
LIN {X 0.070,Y -639.986,Z 1012.612,A 0.000,B 0.000,C 90.000,E1 326.135} C_DIS
LIN {X 0.045,Y -640.789,Z 1012.606,A 0.000,B 0.000,C 90.000,E1 325.135} C_DIS
LIN {X 0.237,Y -641.403,Z 1012.601,A 0.000,B 0.000,C 90.000,E1 324.116} C_DIS
LIN {X -0.020,Y -641.973,Z 1012.592,A 0.000,B 0.000,C 90.000,E1 322.637} C_DIS
LIN {X -0.076,Y -642.505,Z 1012.581,A 0.000,B 0.000,C 90.000,E1 320.642} C_DIS
LIN {X -0.282,Y -643.537,Z 1012.568,A 0.000,B 0.000,C 90.000,E1 318.162} C_DIS
LIN {X -0.184,Y -644.132,Z 1012.561,A 0.000,B 0.000,C 90.000,E1 316.905} C_DIS
LIN {X -0.214,Y -644.986,Z 1012.551,A 0.000,B 0.000,C 90.000,E1 315.162} C_DIS
LIN {X 0.221,Y -646.024,Z 1012.541,A 0.000,B 0.000,C 90.000,E1 313.380} C_DIS
LIN {X -0.079,Y -646.751,Z 1012.534,A 0.000,B 0.000,C 90.000,E1 312.162} C_DIS
LIN {X -0.003,Y -647.566,Z 1012.525,A 0.000,B 0.000,C 90.000,E1 310.415} C_DIS
LIN {X 0.155,Y -648.123,Z 1012.516,A 0.000,B 0.000,C 90.000,E1 308.910} C_DIS
LIN {X -0.013,Y -648.566,Z 1012.509,A 0.000,B 0.000,C 90.000,E1 307.684} C_DIS
LIN {X -0.260,Y -648.920,Z 1012.501,A 0.000,B 0.000,C 90.000,E1 306.217} C_DIS
LIN {X 0.098,Y -649.138,Z 1012.494,A 0.000,B 0.000,C 90.000,E1 304.945} C_DIS
LIN {X 0.127,Y -650.390,Z 1012.476,A 0.000,B 0.000,C 90.000,E1 301.720} C_DIS
LIN {X 0.224,Y -653.075,Z 1012.460,A 0.000,B 0.000,C 90.000,E1 298.743} C_DIS
LIN {X 0.044,Y -655.796,Z 1012.448,A 0.000,B 0.000,C 90.000,E1 296.539} C_DIS
LIN {X -0.251,Y -657.295,Z 1012.441,A 0.000,B 0.000,C 90.000,E1 295.335} C_DIS
LIN {X -0.045,Y -658.186,Z 1012.435,A 0.000,B 0.000,C 90.000,E1 294.335} C_DIS
LIN {X 0.178,Y -658.774,Z 1012.430,A 0.000,B 0.000,C 90.000,E1 293.334} C_DIS
LIN {X -0.204,Y -658.941,Z 1012.424,A 0.000,B 0.000,C 90.000,E1 292.386} C_DIS
LIN {X -0.101,Y -658.707,Z 1012.420,A 0.000,B 0.000,C 90.000,E1 291.642} C_DIS
LIN {X -0.115,Y -657.859,Z 1012.417,A 0.000,B 0.000,C 90.000,E1 291.153} C_DIS
LIN {X -0.239,Y -657.290,Z 1012.416,A 0.000,B 0.000,C 90.000,E1 290.918} C_DIS
LIN {X -0.206,Y -654.348,Z 1012.413,A 0.000,B 0.000,C 90.000,E1 290.301} C_DIS
LIN {X -0.156,Y -653.359,Z 1012.412,A 0.000,B 0.000,C 90.000,E1 290.174} C_DIS
LIN {X -0.335,Y -652.192,Z 1012.411,A 0.000,B 0.000,C 90.000,E1 290.066} C_DIS
LIN {X -0.287,Y -650.811,Z 1012.411,A 0.000,B 0.000,C 90.000,E1 289.939} C_DIS
LIN {X -0.022,Y -647.830,Z 1012.409,A 0.000,B 0.000,C 90.000,E1 289.685} C_DIS
LIN {X -0.008,Y -646.307,Z 1012.409,A 0.000,B 0.000,C 90.000,E1 289.577} C_DIS
LIN {X -0.209,Y -640.023,Z 1012.407,A 0.000,B 0.000,C 90.000,E1 289.214} C_DIS
LIN {X -0.246,Y -629.987,Z 1012.404,A 0.000,B 0.000,C 90.000,E1 288.725} C_DIS
LIN {X 0.065,Y -626.403,Z 1012.403,A 0.000,B 0.000,C 90.000,E1 288.489} C_DIS
LIN {X 0.003,Y -626.379,Z 1012.403,A 0.000,B 0.000,C 90.000,E1 288.489} C_DIS
LIN {X 0.024,Y -627.020,Z 1012.402,A 0.000,B 0.000,C 90.000,E1 288.308} C_DIS
LIN {X -0.190,Y -629.540,Z 1012.400,A 0.000,B 0.000,C 90.000,E1 287.946} C_DIS
LIN {X -0.199,Y -631.144,Z 1012.398,A 0.000,B 0.000,C 90.000,E1 287.692} C_DIS
LIN {X -0.021,Y -633.641,Z 1012.396,A 0.000,B 0.000,C 90.000,E1 287.330} C_DIS
LIN {X -0.253,Y -637.729,Z 1012.393,A 0.000,B 0.000,C 90.000,E1 286.732} C_DIS
LIN {X -0.123,Y -641.980,Z 1012.389,A 0.000,B 0.000,C 90.000,E1 285.969} C_DIS
LIN {X -0.262,Y -644.404,Z 1012.386,A 0.000,B 0.000,C 90.000,E1 285.481} C_DIS
LIN {X 0.060,Y -646.455,Z 1012.383,A 0.000,B 0.000,C 90.000,E1 284.954} C_DIS
LIN {X -0.365,Y -648.702,Z 1012.379,A 0.000,B 0.000,C 90.000,E1 284.245} C_DIS
LIN {X -0.004,Y -649.941,Z 1012.376,A 0.000,B 0.000,C 90.000,E1 283.716} C_DIS
LIN {X -0.265,Y -650.705,Z 1012.373,A 0.000,B 0.000,C 90.000,E1 283.244} C_DIS
LIN {X -0.014,Y -651.462,Z 1012.369,A 0.000,B 0.000,C 90.000,E1 282.479} C_DIS
LIN {X 0.242,Y -651.626,Z 1012.365,A 0.000,B 0.000,C 90.000,E1 281.715} C_DIS
LIN {X -0.015,Y -651.368,Z 1012.362,A 0.000,B 0.000,C 90.000,E1 281.243} C_DIS
LIN {X 0.242,Y -650.908,Z 1012.360,A 0.000,B 0.000,C 90.000,E1 280.725} C_DIS
LIN {X -0.021,Y -650.115,Z 1012.357,A 0.000,B 0.000,C 90.000,E1 280.254} C_DIS
LIN {X -0.156,Y -649.636,Z 1012.356,A 0.000,B 0.000,C 90.000,E1 280.018} C_DIS
LIN {X 0.097,Y -648.395,Z 1012.353,A 0.000,B 0.000,C 90.000,E1 279.500} C_DIS
LIN {X -0.190,Y -646.751,Z 1012.350,A 0.000,B 0.000,C 90.000,E1 279.029} C_DIS
LIN {X 0.048,Y -644.686,Z 1012.347,A 0.000,B 0.000,C 90.000,E1 278.511} C_DIS
LIN {X 0.277,Y -642.124,Z 1012.345,A 0.000,B 0.000,C 90.000,E1 277.992} C_DIS
LIN {X 0.109,Y -640.723,Z 1012.343,A 0.000,B 0.000,C 90.000,E1 277.757} C_DIS
LIN {X 0.305,Y -637.328,Z 1012.340,A 0.000,B 0.000,C 90.000,E1 277.239} C_DIS
LIN {X -0.016,Y -634.304,Z 1012.338,A 0.000,B 0.000,C 90.000,E1 276.891} C_DIS
LIN {X 0.137,Y -629.752,Z 1012.336,A 0.000,B 0.000,C 90.000,E1 276.372} C_DIS
LIN {X -0.144,Y -627.374,Z 1012.334,A 0.000,B 0.000,C 90.000,E1 276.144} C_DIS
LIN {X 0.148,Y -620.859,Z 1012.331,A 0.000,B 0.000,C 90.000,E1 275.511} C_DIS
LIN {X 0.164,Y -615.219,Z 1012.328,A 0.000,B 0.000,C 90.000,E1 275.049} C_DIS
LIN {X -0.237,Y -610.583,Z 1012.326,A 0.000,B 0.000,C 90.000,E1 274.759} C_DIS
LIN {X 0.179,Y -606.021,Z 1012.325,A 0.000,B 0.000,C 90.000,E1 274.416} C_DIS
LIN {X -0.160,Y -599.461,Z 1012.323,A 0.000,B 0.000,C 90.000,E1 274.073} C_DIS
LIN {X -0.059,Y -592.491,Z 1012.321,A 0.000,B 0.000,C 90.000,E1 273.726} C_DIS
LIN {X -0.003,Y -585.335,Z 1012.319,A 0.000,B 0.000,C 90.000,E1 273.440} C_DIS
LIN {X -0.118,Y -578.780,Z 1012.318,A 0.000,B 0.000,C 90.000,E1 273.269} C_DIS
LIN {X -0.125,Y -571.269,Z 1012.317,A 0.000,B 0.000,C 90.000,E1 273.094} C_DIS
LIN {X 0.040,Y -565.632,Z 1012.317,A 0.000,B 0.000,C 90.000,E1 272.980} C_DIS
LIN {X 0.098,Y -558.472,Z 1012.316,A 0.000,B 0.000,C 90.000,E1 272.922} C_DIS
LIN {X 0.047,Y -543.892,Z 1012.316,A 0.000,B 0.000,C 90.000,E1 272.922} C_DIS
LIN {X 0.238,Y -542.981,Z 1012.315,A 0.000,B 0.000,C 90.000,E1 272.751} C_DIS
LIN {X 0.241,Y -542.465,Z 1012.314,A 0.000,B 0.000,C 90.000,E1 272.407} C_DIS
LIN {X -0.245,Y -541.967,Z 1012.310,A 0.000,B 0.000,C 90.000,E1 271.892} C_DIS
LIN {X -0.079,Y -540.937,Z 1012.301,A 0.000,B 0.000,C 90.000,E1 270.172} C_DIS
LIN {X 0.031,Y -540.036,Z 1012.293,A 0.000,B 0.000,C 90.000,E1 268.740} C_DIS
LIN {X 0.119,Y -539.227,Z 1012.287,A 0.000,B 0.000,C 90.000,E1 267.593} C_DIS
LIN {X 0.257,Y -537.677,Z 1012.276,A 0.000,B 0.000,C 90.000,E1 265.584} C_DIS
LIN {X -0.135,Y -536.374,Z 1012.266,A 0.000,B 0.000,C 90.000,E1 263.913} C_DIS
LIN {X -0.008,Y -535.137,Z 1012.258,A 0.000,B 0.000,C 90.000,E1 262.470} C_DIS
LIN {X 0.091,Y -533.733,Z 1012.250,A 0.000,B 0.000,C 90.000,E1 261.027} C_DIS
LIN {X 0.282,Y -532.485,Z 1012.244,A 0.000,B 0.000,C 90.000,E1 259.859} C_DIS
LIN {X -0.009,Y -529.937,Z 1012.231,A 0.000,B 0.000,C 90.000,E1 257.589} C_DIS
LIN {X -0.240,Y -528.417,Z 1012.223,A 0.000,B 0.000,C 90.000,E1 256.172} C_DIS
LIN {X 0.185,Y -526.134,Z 1012.212,A 0.000,B 0.000,C 90.000,E1 254.102} C_DIS
LIN {X 0.022,Y -524.572,Z 1012.204,A 0.000,B 0.000,C 90.000,E1 252.670} C_DIS
LIN {X -0.014,Y -522.979,Z 1012.196,A 0.000,B 0.000,C 90.000,E1 251.221} C_DIS
LIN {X 0.097,Y -521.106,Z 1012.188,A 0.000,B 0.000,C 90.000,E1 249.752} C_DIS
LIN {X -0.012,Y -518.452,Z 1012.176,A 0.000,B 0.000,C 90.000,E1 247.720} C_DIS
LIN {X 0.075,Y -516.854,Z 1012.170,A 0.000,B 0.000,C 90.000,E1 246.538} C_DIS
LIN {X -0.207,Y -514.756,Z 1012.162,A 0.000,B 0.000,C 90.000,E1 245.101} C_DIS
LIN {X -0.084,Y -513.463,Z 1012.157,A 0.000,B 0.000,C 90.000,E1 244.204} C_DIS
LIN {X 0.120,Y -510.605,Z 1012.147,A 0.000,B 0.000,C 90.000,E1 242.410} C_DIS
LIN {X -0.201,Y -507.707,Z 1012.137,A 0.000,B 0.000,C 90.000,E1 240.667} C_DIS
LIN {X -0.036,Y -505.644,Z 1012.130,A 0.000,B 0.000,C 90.000,E1 239.459} C_DIS
LIN {X 0.221,Y -503.991,Z 1012.125,A 0.000,B 0.000,C 90.000,E1 238.535} C_DIS
LIN {X 0.084,Y -500.477,Z 1012.115,A 0.000,B 0.000,C 90.000,E1 236.755} C_DIS
LIN {X 0.130,Y -497.807,Z 1012.109,A 0.000,B 0.000,C 90.000,E1 235.548} C_DIS
LIN {X -0.268,Y -495.713,Z 1012.104,A 0.000,B 0.000,C 90.000,E1 234.689} C_DIS
LIN {X 0.012,Y -493.531,Z 1012.099,A 0.000,B 0.000,C 90.000,E1 233.749} C_DIS
LIN {X 0.200,Y -489.078,Z 1012.089,A 0.000,B 0.000,C 90.000,E1 231.904} C_DIS
LIN {X 0.015,Y -484.111,Z 1012.077,A 0.000,B 0.000,C 90.000,E1 229.784} C_DIS
LIN {X -0.046,Y -479.184,Z 1012.065,A 0.000,B 0.000,C 90.000,E1 227.634} C_DIS
LIN {X -0.252,Y -474.565,Z 1012.053,A 0.000,B 0.000,C 90.000,E1 225.486} C_DIS
LIN {X 0.242,Y -471.426,Z 1012.044,A 0.000,B 0.000,C 90.000,E1 223.866} C_DIS
LIN {X 0.171,Y -466.793,Z 1012.032,A 0.000,B 0.000,C 90.000,E1 221.676} C_DIS
LIN {X 0.215,Y -463.426,Z 1012.023,A 0.000,B 0.000,C 90.000,E1 220.092} C_DIS
LIN {X 0.157,Y -460.596,Z 1012.016,A 0.000,B 0.000,C 90.000,E1 218.830} C_DIS
LIN {X -0.116,Y -456.308,Z 1012.005,A 0.000,B 0.000,C 90.000,E1 216.950} C_DIS
LIN {X -0.122,Y -452.128,Z 1011.995,A 0.000,B 0.000,C 90.000,E1 215.025} C_DIS
LIN {X 0.026,Y -446.437,Z 1011.980,A 0.000,B 0.000,C 90.000,E1 212.418} C_DIS
LIN {X 0.081,Y -441.457,Z 1011.967,A 0.000,B 0.000,C 90.000,E1 210.129} C_DIS
LIN {X 0.046,Y -438.547,Z 1011.960,A 0.000,B 0.000,C 90.000,E1 208.821} C_DIS
LIN {X -0.035,Y -435.503,Z 1011.953,A 0.000,B 0.000,C 90.000,E1 207.513} C_DIS
LIN {X -0.154,Y -431.029,Z 1011.942,A 0.000,B 0.000,C 90.000,E1 205.540} C_DIS
LIN {X 0.209,Y -427.254,Z 1011.933,A 0.000,B 0.000,C 90.000,E1 203.823} C_DIS
LIN {X 0.059,Y -421.383,Z 1011.918,A 0.000,B 0.000,C 90.000,E1 201.153} C_DIS
LIN {X -0.106,Y -417.313,Z 1011.906,A 0.000,B 0.000,C 90.000,E1 199.141} C_DIS
LIN {X -0.104,Y -413.546,Z 1011.895,A 0.000,B 0.000,C 90.000,E1 197.094} C_DIS
LIN {X 0.103,Y -409.548,Z 1011.882,A 0.000,B 0.000,C 90.000,E1 194.662} C_DIS
LIN {X 0.113,Y -405.422,Z 1011.866,A 0.000,B 0.000,C 90.000,E1 191.895} C_DIS
LIN {X -0.175,Y -403.618,Z 1011.859,A 0.000,B 0.000,C 90.000,E1 190.546} C_DIS
LIN {X -0.169,Y -402.690,Z 1011.853,A 0.000,B 0.000,C 90.000,E1 189.500} C_DIS
LIN {X -0.172,Y -402.458,Z 1011.849,A 0.000,B 0.000,C 90.000,E1 188.803} C_DIS
LIN {X -0.143,Y -402.522,Z 1011.848,A 0.000,B 0.000,C 90.000,E1 188.624} C_DIS
LIN {X -0.179,Y -403.032,Z 1011.845,A 0.000,B 0.000,C 90.000,E1 188.106} C_DIS
LIN {X -0.182,Y -403.204,Z 1011.843,A 0.000,B 0.000,C 90.000,E1 187.757} C_DIS
LIN {X -0.185,Y -403.645,Z 1011.841,A 0.000,B 0.000,C 90.000,E1 187.409} C_DIS
LIN {X 0.020,Y -405.135,Z 1011.838,A 0.000,B 0.000,C 90.000,E1 186.777} C_DIS
LIN {X 0.048,Y -408.104,Z 1011.834,A 0.000,B 0.000,C 90.000,E1 186.030} C_DIS
LIN {X 0.043,Y -412.369,Z 1011.829,A 0.000,B 0.000,C 90.000,E1 185.277} C_DIS
LIN {X 0.067,Y -417.255,Z 1011.826,A 0.000,B 0.000,C 90.000,E1 184.588} C_DIS
LIN {X 0.064,Y -429.687,Z 1011.817,A 0.000,B 0.000,C 90.000,E1 183.094} C_DIS
LIN {X -0.108,Y -439.458,Z 1011.811,A 0.000,B 0.000,C 90.000,E1 182.007} C_DIS
LIN {X -0.166,Y -450.234,Z 1011.804,A 0.000,B 0.000,C 90.000,E1 180.745} C_DIS
LIN {X -0.122,Y -456.898,Z 1011.800,A 0.000,B 0.000,C 90.000,E1 179.943} C_DIS
LIN {X 0.050,Y -464.782,Z 1011.794,A 0.000,B 0.000,C 90.000,E1 178.969} C_DIS
LIN {X 0.178,Y -471.140,Z 1011.790,A 0.000,B 0.000,C 90.000,E1 178.165} C_DIS
LIN {X 0.146,Y -478.421,Z 1011.785,A 0.000,B 0.000,C 90.000,E1 177.249} C_DIS
LIN {X 0.239,Y -481.953,Z 1011.782,A 0.000,B 0.000,C 90.000,E1 176.788} C_DIS
LIN {X 0.010,Y -487.730,Z 1011.778,A 0.000,B 0.000,C 90.000,E1 176.045} C_DIS
LIN {X -0.030,Y -496.254,Z 1011.771,A 0.000,B 0.000,C 90.000,E1 174.837} C_DIS
LIN {X -0.224,Y -502.327,Z 1011.766,A 0.000,B 0.000,C 90.000,E1 173.970} C_DIS
LIN {X 0.043,Y -510.062,Z 1011.760,A 0.000,B 0.000,C 90.000,E1 172.761} C_DIS
LIN {X -0.144,Y -515.580,Z 1011.755,A 0.000,B 0.000,C 90.000,E1 171.894} C_DIS
LIN {X -0.166,Y -518.272,Z 1011.753,A 0.000,B 0.000,C 90.000,E1 171.489} C_DIS
LIN {X 0.030,Y -524.123,Z 1011.747,A 0.000,B 0.000,C 90.000,E1 170.443} C_DIS
LIN {X -0.237,Y -528.423,Z 1011.743,A 0.000,B 0.000,C 90.000,E1 169.746} C_DIS
LIN {X -0.182,Y -536.101,Z 1011.736,A 0.000,B 0.000,C 90.000,E1 168.465} C_DIS
LIN {X -0.177,Y -545.991,Z 1011.726,A 0.000,B 0.000,C 90.000,E1 166.756} C_DIS
LIN {X 0.174,Y -557.023,Z 1011.715,A 0.000,B 0.000,C 90.000,E1 164.755} C_DIS
LIN {X 0.207,Y -563.680,Z 1011.708,A 0.000,B 0.000,C 90.000,E1 163.504} C_DIS
LIN {X -0.203,Y -570.104,Z 1011.702,A 0.000,B 0.000,C 90.000,E1 162.308} C_DIS
LIN {X -0.250,Y -575.626,Z 1011.696,A 0.000,B 0.000,C 90.000,E1 161.221} C_DIS
LIN {X 0.164,Y -581.995,Z 1011.688,A 0.000,B 0.000,C 90.000,E1 159.826} C_DIS
LIN {X -0.065,Y -586.824,Z 1011.682,A 0.000,B 0.000,C 90.000,E1 158.773} C_DIS
LIN {X -0.227,Y -591.371,Z 1011.676,A 0.000,B 0.000,C 90.000,E1 157.720} C_DIS
LIN {X 0.217,Y -595.541,Z 1011.670,A 0.000,B 0.000,C 90.000,E1 156.613} C_DIS
LIN {X -0.054,Y -598.491,Z 1011.666,A 0.000,B 0.000,C 90.000,E1 155.845} C_DIS
LIN {X -0.068,Y -602.091,Z 1011.660,A 0.000,B 0.000,C 90.000,E1 154.793} C_DIS
LIN {X -0.330,Y -605.373,Z 1011.654,A 0.000,B 0.000,C 90.000,E1 153.768} C_DIS
LIN {X 0.228,Y -609.191,Z 1011.647,A 0.000,B 0.000,C 90.000,E1 152.410} C_DIS
LIN {X -0.011,Y -613.565,Z 1011.638,A 0.000,B 0.000,C 90.000,E1 150.873} C_DIS
LIN {X 0.195,Y -615.635,Z 1011.634,A 0.000,B 0.000,C 90.000,E1 150.078} C_DIS
LIN {X 0.147,Y -619.773,Z 1011.625,A 0.000,B 0.000,C 90.000,E1 148.535} C_DIS
LIN {X 0.180,Y -623.800,Z 1011.617,A 0.000,B 0.000,C 90.000,E1 146.993} C_DIS
LIN {X -0.060,Y -628.436,Z 1011.607,A 0.000,B 0.000,C 90.000,E1 145.229} C_DIS
LIN {X -0.034,Y -632.378,Z 1011.598,A 0.000,B 0.000,C 90.000,E1 143.703} C_DIS
LIN {X 0.053,Y -635.647,Z 1011.591,A 0.000,B 0.000,C 90.000,E1 142.431} C_DIS
LIN {X -0.026,Y -639.548,Z 1011.583,A 0.000,B 0.000,C 90.000,E1 140.928} C_DIS
LIN {X -0.024,Y -643.959,Z 1011.573,A 0.000,B 0.000,C 90.000,E1 139.175} C_DIS
LIN {X 0.015,Y -647.664,Z 1011.565,A 0.000,B 0.000,C 90.000,E1 137.676} C_DIS
LIN {X -0.074,Y -655.009,Z 1011.550,A 0.000,B 0.000,C 90.000,E1 134.960} C_DIS
LIN {X 0.139,Y -661.055,Z 1011.539,A 0.000,B 0.000,C 90.000,E1 132.975} C_DIS
LIN {X 0.068,Y -666.542,Z 1011.529,A 0.000,B 0.000,C 90.000,E1 131.272} C_DIS
LIN {X -0.325,Y -670.381,Z 1011.523,A 0.000,B 0.000,C 90.000,E1 130.092} C_DIS
LIN {X -0.120,Y -674.600,Z 1011.515,A 0.000,B 0.000,C 90.000,E1 128.624} C_DIS
LIN {X -0.379,Y -678.051,Z 1011.508,A 0.000,B 0.000,C 90.000,E1 127.443} C_DIS
LIN {X 0.109,Y -681.989,Z 1011.500,A 0.000,B 0.000,C 90.000,E1 125.964} C_DIS
LIN {X 0.107,Y -685.260,Z 1011.493,A 0.000,B 0.000,C 90.000,E1 124.771} C_DIS
LIN {X 0.152,Y -688.344,Z 1011.487,A 0.000,B 0.000,C 90.000,E1 123.579} C_DIS
LIN {X 0.092,Y -692.520,Z 1011.477,A 0.000,B 0.000,C 90.000,E1 121.926} C_DIS
LIN {X -0.153,Y -694.853,Z 1011.472,A 0.000,B 0.000,C 90.000,E1 121.003} C_DIS
LIN {X 0.339,Y -696.490,Z 1011.468,A 0.000,B 0.000,C 90.000,E1 120.256} C_DIS
LIN {X -0.111,Y -697.936,Z 1011.464,A 0.000,B 0.000,C 90.000,E1 119.589} C_DIS
LIN {X -0.026,Y -699.837,Z 1011.458,A 0.000,B 0.000,C 90.000,E1 118.409} C_DIS
LIN {X -0.166,Y -700.678,Z 1011.454,A 0.000,B 0.000,C 90.000,E1 117.719} C_DIS
LIN {X -0.154,Y -702.197,Z 1011.444,A 0.000,B 0.000,C 90.000,E1 115.848} C_DIS
LIN {X 0.026,Y -702.873,Z 1011.438,A 0.000,B 0.000,C 90.000,E1 114.899} C_DIS
LIN {X -0.066,Y -703.046,Z 1011.435,A 0.000,B 0.000,C 90.000,E1 114.207} C_DIS
LIN {X -0.436,Y -702.402,Z 1011.432,A 0.000,B 0.000,C 90.000,E1 113.770} C_DIS
LIN {X -0.158,Y -701.997,Z 1011.431,A 0.000,B 0.000,C 90.000,E1 113.515} C_DIS
LIN {X 0.116,Y -701.035,Z 1011.429,A 0.000,B 0.000,C 90.000,E1 113.259} C_DIS
LIN {X 0.247,Y -699.275,Z 1011.427,A 0.000,B 0.000,C 90.000,E1 112.898} C_DIS
LIN {X -0.263,Y -698.553,Z 1011.427,A 0.000,B 0.000,C 90.000,E1 112.823} C_DIS
LIN {X -0.133,Y -697.475,Z 1011.426,A 0.000,B 0.000,C 90.000,E1 112.695} C_DIS
LIN {X 0.054,Y -694.363,Z 1011.425,A 0.000,B 0.000,C 90.000,E1 112.461} C_DIS
LIN {X 0.307,Y -689.752,Z 1011.423,A 0.000,B 0.000,C 90.000,E1 112.153} C_DIS
LIN {X -0.292,Y -684.657,Z 1011.422,A 0.000,B 0.000,C 90.000,E1 112.025} C_DIS
LIN {X -0.108,Y -677.221,Z 1011.422,A 0.000,B 0.000,C 90.000,E1 111.897} C_DIS
LIN {X 0.252,Y -675.445,Z 1011.422,A 0.000,B 0.000,C 90.000,E1 111.844} C_DIS
LIN {X 0.183,Y -617.109,Z 1011.422,A 0.000,B 0.000,C 90.000,E1 111.844} C_DIS
LIN {X -0.168,Y -610.880,Z 1011.421,A 0.000,B 0.000,C 90.000,E1 111.716} C_DIS
LIN {X -0.047,Y -604.446,Z 1011.419,A 0.000,B 0.000,C 90.000,E1 111.461} C_DIS
LIN {X -0.130,Y -600.208,Z 1011.418,A 0.000,B 0.000,C 90.000,E1 111.280} C_DIS
LIN {X -0.023,Y -594.168,Z 1011.416,A 0.000,B 0.000,C 90.000,E1 110.918} C_DIS
